(* Logix 5000 project; controller cal1615 1756-L62 rev 20.19; software revision 20.05; part 7 of 81 *)

   p23r11_permissive_jog : BOOL := 1;   // Impreg Servo Operator Side Perimssive Jog
   p23r11_pos_offset : REAL := 0.0005;
   p23r11_request_jog_fwd : BOOL;   // Impreg Servo Operator Side Requset Jog Forward
   p23r11_request_jog_rev : BOOL;   // Impreg Servo Operator Side Requset Jog Reverse
   p23r11_request_position : BOOL;   // Impreg Servo Operator Side Request Position
   p23r11_request_start : BOOL;   // Impreg Servo Operator Side Request Start
   p23r11_request_zero : BOOL;   // Impreg Servo Operator Side Request Zero
   p23r11_selected_position : REAL := 0.016;
   p23r11_servo_not_ready : BOOL;   // Impreg Servo Operator Side Not Ready
   p23r11_servo_status_ab : BOOL := 1;   // Impreg Servo Operator Side AB Status
   p23r11_servo_status_af : BOOL;   // Impreg Servo Operator Side AF Status
   p23r11_servo_status_bb : BOOL;   // Impreg Servo Operator Side BB Status
   p23r11_step_4_dwell : TIMER := (PRE := 1000);
   p23r11_timer : TIMER[4] := ([0].ACC := 33, [0].EN := 1, [0].DN := 1);   // Impreg Servo Operator Side Timer
   p23r11_timer_fault : TIMER[4];   // Impreg Servo Drive Side Fault Delay
   p23r11_timer_warning : TIMER[4];   // Impreg Servo Drive Side Warning Delay
   p23r12 : routine := (comment := -1073741570, state := 3);   // Impreg Servo Drive Side
        .FAULT.0   // Impreg Servo Drive Side Operating Mode Error
        .FAULT.1   // Impreg Servo Drive Side Servo Fault
        .FAULT.3   // Tension Stand 2 VFD Not in Network Mode
        .WARNING.0   // Impreg Servo Drive Side Servo Warning
        .WARNING.1   // Tension Stand 2 VFD Motor Thermistor Not OK
        .WARNING.2   // Tension Stand 2 VFD Motor Blower Not Running
        .WARNING.3   // Tension Stand 2 VFD Brake Thermistor Not Ok
        .UNACK_FAULT   // Impreg Servo Drive Side Unacknoledged Faults Exist
        .UNACK_WARNING   // Impreg Servo Drive Side Unack. Warnings Exist
   p23r12_gap_sequence_enabled : BOOL;
   p23r12_impreg_gap_ds : REAL := 0.016;
   p23r12_offsets : REAL[100] := ([5] := -0.0005, [8] := 0.00015, [10] := -0.0002);
   p23r12_permissive_jog : BOOL := 1;   // Impreg Servo Drive Side Perimssive Jog
   p23r12_pos_offset : REAL;
   p23r12_request_jog_fwd : BOOL;   // Impreg Servo Drive Side Requset Jog Forward
   p23r12_request_jog_rev : BOOL;   // Impreg Servo Drive Side Requset Jog Reverse
   p23r12_request_position : BOOL;   // Impreg Servo Drive Side Request Position
   p23r12_request_start : BOOL;   // Caoter Servo Drive Side Start Request
   p23r12_request_zero : BOOL;   // Impreg Servo Drive Side Request Zero
   p23r12_selected_position : REAL := 0.016;
   p23r12_servo_not_ready : BOOL;   // Impreg Servo Drive Side Not Ready
   p23r12_servo_status_ab : BOOL := 1;   // Impreg Servo Drive Side AB Status
   p23r12_servo_status_af : BOOL;   // Impreg Servo Drive Side AF Status
   p23r12_servo_status_bb : BOOL;   // Impreg Servo Drive Side BB Status
   p23r12_step_4_dwell : TIMER := (PRE := 1000);
   p23r12_timer : TIMER[4] := ([0].ACC := 33, [0].EN := 1, [0].DN := 1);   // Impreg Servo Drive Side Timer
   p23r12_timer_fault : TIMER[4];   // Impreg Servo Drive Side Fault Delay
   p23r12_timer_warning : TIMER[4];   // Impreg Servo Drive Side Warning Delay
   p23r13 : routine := (comment := -1073741697, oneshot := 3);
        .FAULT.0   // Impreg Supply VFD Drive Faulted
        .FAULT.2   // Impreg Supply VFD Drive Not Ready
        .FAULT.3   // Impreg Supply VFD Not in Remote Mode
        .FAULT.4   // Impreg Supply VFD Motor Temperature
        .FAULT_ACK   // Impreg Static Control 2 Faults
        .WARNING.0   // Impreg Supply Fan VFD Drive Warning
        .WARNING.1   // Impreg Supply Fan VFD Supply Filter Dirty
        .WARNING_ACK   // Impreg Static Control 2 Warnings
        .UNACK_FAULT   // Impreg Static Control 2 Unack. Faults Exist
        .UNACK_WARNING   // Impreg Static Control 2 Unack. Warnings Exist
   p23r13_pb_start : BOOL;   // Impreg Supply VFD Start
   p23r13_pb_stop : BOOL;   // Impreg Supply VFD Stop
   p23r13_request_auto_run : BOOL;   // Impreg Supply Fan VFD Request Auto Run
   p23r13_run_permissive : BOOL := 1;   // Impreg Supply VFD Run Permissive
   p23r13_timer_fault : TIMER[10] := ([5].PRE := 5000);   // Impreg Supply VFD Fault Dwell Timer
   p23r13_timer_warning : TIMER[4] := ([1].PRE := 1000, [2].PRE := 10000);   // Impreg Supply VFD Warning Dwell Timer
   p23r13_vfd_stopped : BOOL := 1;   // Impreg Supply VFD Stopped
   p23r15 : routine := (comment := -1073741713, warning := 1, unack_warning := 1);   // Impreg Metering Roll VFD
        .FAULT.0   // Impreg Metering Roll VFD Drive Fault
        .FAULT.2   // Impreg Metering Roll VFD Not Ready
        .FAULT.3   // Impreg Metering Roll VFD Not in Network Mode
        .FAULT.4   // Impreg Metering Roll VFD Motor Temperature Failure
        .WARNING.0   // Impreg Metering VFD Drive Warning
        .WARNING.1   // Impreg Metering Roll VFD Motor Thermistor Not OK
        .WARNING.2   // Impreg Metering Roll VFD Motor Blower Not Running
        .WARNING.3   // Impreg Metering Roll VFD Brake Thermistor Not Ok
        .UNACK_FAULT   // Impreg Metering Roll VFD Unacknoledged Faults Exists
        .UNACK_WARNING   // Impreg Metering Roll VFD Unacknoledged Warning Exists
   p23r15_acc_decel_ramp : SYS_ACC_DEC_RAMP := (IN_param_master_accel_rate := 15.0, IN_param_master_decel_rate := 15.0, IN_last_scan_s := 0.033662);   // Impreg Metering Roll VFD Accel/Decel Ramp
   p23r15_adjust_dwell1 : TIMER := (PRE := 20000);   // Impreg Metering Roll VFD Adjustment Dwell Timer
   p23r15_average_tension : REAL := 87.4577;   // Impreg Metering Roll VFD Average Tension
   p23r15_dead_band_minus : REAL := 45.0;   // Impreg Metering Roll VFD Dead Band -
   p23r15_dead_band_plus : REAL := 55.0;   // Impreg Metering Roll VFD Dead Band +
   p23r15_dead_band_setpoint : REAL := 5.0;
   p23r15_debounce_timer : TIMER := (PRE := 2000, EN := 1, DN := 1);   // Impreg Metering Roll VFD Tension Ok Debounce Timer
   p23r15_ffl : CONTROL := (LEN := 10, POS := 9);   // Impreg Metering Roll VFD Avererage FFL
   p23r15_ffu_temp : REAL := 102.55185;
   p23r15_fll_stack : REAL[50] := ([0] := 98.387886, [1] := 74.37622, [2] := 97.50486, [3] := 91.988014, [4] := 72.294235, [5] := 89.74401, [6] := 102.07388, [7] := 75.97214, [8] := 84.77803, [10] := 108.79131, [11] := 101.68503, [12] := 100.24141, [13] := 100.53305, [14] := 105.432594, [15] := 103.07518, [16] := 106.29294, [17] := 103.507774, [18] := 102.11763, [20] := 103.94038, [21] := 99.57064, [22] := 100.149055, [23] := 101.106606, [24] := 99.040825, [25] := 99.71646, [26] := 98.370056, [27] := 101.34964, [28] := 96.83409, [29] := 100.43584, [30] := 96.83409, [31] := 98.60823, [32] := 99.90603, [33] := 99.76507, [34] := 101.53921, [35] := 98.60823, [36] := 102.02042, [37] := 100.917046, [38] := 106.676926);
   p23r15_mean_adjust_acitve : BOOL;   // Impreg Metering Roll VFD Mean Adjust Active
   p23r15_minus_adjust : REAL := 1.0;
   p23r15_minus_adjust_acitve : BOOL;   // Impreg Metering Roll VFD Minus Adjust Active
   p23r15_minus_offset : REAL := -0.48000002;
   p23r15_neutral_offset : REAL := 0.4;
   p23r15_permissive_jog : BOOL := 1;   // Impreg Impreg VFD Permissive Jog
   p23r15_permissive_run : BOOL := 1;   // Impreg Metering Roll VFD Permissive Run
   p23r15_pid_tension_control : BOOL := 1;   // Impreg Metering Roll VFD PID Wet Web Active
   p23r15_plus_adjust : REAL := 1.0;
   p23r15_plus_adjust_acitve : BOOL;   // Impreg Plus Adjust Active
   p23r15_plus_offset : REAL := 4.7999997;
   p23r15_request_jog_fwd : BOOL;   // Impreg Metering Roll VFD Request Jog FWD
   p23r15_request_jog_rev : BOOL;   // Impreg Metering Roll VFD Request Jog REV
   p23r15_request_line_run : BOOL;   // Impreg Metering Roll VFD Request Line Run
   p23r15_request_thread_fwd : BOOL;   // Impreg Metering Roll VFD Request Thread FWD
   p23r15_request_thread_rev : BOOL;   // Impreg Metering Roll VFD Request Thread REV
   p23r15_sample_timer : TIMER := (PRE := 100);   // Impreg Metering Roll Sample Timer
   p23r15_selected_speed : REAL;   // Impreg Metering Roll VFD Selected Speed
   p23r15_timer_fault : TIMER[10];   // Impreg Pick Up Roll VFD Fault Timer
   p23r15_timer_warning : TIMER[5];   // Impreg Pick Up Roll VFD Warning Timer
   p23r15_ts1_tension_ok : BOOL := 1;   // Impreg Metering Roll VFD TS 1 Tension Ok
   p23r15_zero_speed : BOOL := 1;   // Impreg Metering Roll VFD At Zero Speed
   p23r17_adjusted_speed : REAL;
   p23r17_di_brake : BOOL;
   p23r17_di_therm : BOOL;
   p23r17_permissive_jog : BOOL := 1;
   p23r17_permissive_run : BOOL := 1;
   p23r17_request_jog_fwd : BOOL;
   p23r17_request_thread_fwd : BOOL;
   p23r17_request_thread_rev : BOOL;
   p23r17_selected_speed : REAL;
   p23r17_spd_adj : REAL := -0.5;
   p23r17_sprng_assist_hmi_auto : BOOL;
   p23r17_sprng_assist_hmi_jog : BOOL;
   p23r17_timer_fault : TIMER[10] := ([2].PRE := 3000, [4].ACC := 33, [4].EN := 1, [4].DN := 1, [5].ACC := 33, [5].EN := 1, [5].DN := 1);
   p23r17_timer_warning : TIMER[5];
   p23r17_zero_speed : BOOL := 1;
   p24_di_edge_guide_auto : BOOL := 1;   // Edge Control Inputs SS: Edge Guide Manual/Auto Auto
   p24_di_edge_guide_center : BOOL := 1;   // Edge Control Inputs PB: Edge Guide Center
   p24_di_edge_guide_left : BOOL := 1;   // Edge Control Inputs PB: Edge Guide Left
   p24_di_edge_guide_right : BOOL := 1;   // Edge Control Inputs PB: Edge Guide Right
   p24_dint_to_hmi : DINT[16];
   p24_do_edge_guide_input_1 : BOOL := 1;   // Edge Guide Digital Output Input 1
   p24_do_edge_guide_input_2 : BOOL;   // Edge Guide Digital Output Input 2
   p24_do_edge_guide_input_3 : BOOL;   // Edge Guide Digital Output Input 3
   p24_do_edge_guide_input_4 : BOOL;   // Edge Guide Digital Output Input 4
   p24_do_edge_guide_input_5 : BOOL;   // Edge Guide Digital Output Input 5
   p24_real_to_hmi : REAL[112];   // Tension Stand 2 Real to HMI
   p24r01 : routine := (comment := 7);
   p24r02 : routine := (comment := -1073741761);   // Edge Control Misc Control
        .UNACK_FAULT   // Edge Control Misc Control Unacknowleged Fault Exist
        .UNACK_WARNING   // Edge Control Misc Control Unacknowleged Warning Exist
   p24r02_fault_exists : BOOL;
   p24r02_timer_fault : TIMER[4];   // Edge Control Misc Control Fault Delay
   p24r02_timer_warning : TIMER[4];   // Edge Control Misc Control Warning Delay
   p24r02_unack_fault : BOOL;   // Tension Stand 2 Misc Control Unacknowledged Fault Exists
   p24r02_unack_warning : BOOL;   // Tension Stand 2 Misc Control Unacknowledged Warning Exists
   p24r02_warning_exists : BOOL;
   p24r03 : routine := (comment := -1073741761);   // Edge Control Inputs
        .UNACK_FAULT   // Edge Control Inputs Unacknowleged Fault Exist
        .UNACK_WARNING   // Edge Control Inputs Unacknowleged Warning Exist
   p24r03_timer_fault : TIMER[4];   // Edge Control Inputs Fault Delay
   p24r03_timer_warning : TIMER[4];   // Edge Control Inputs Warning Delay
   p24r04 : routine := (comment := -1073741809);   // Edge Control Outputs
        .UNACK_FAULT   // Edge Control Outputs Unacknowleged Fault Exist
        .UNACK_WARNING   // Edge Control Outputs Unacknowleged Warning Exist
   p24r04_timer_fault : TIMER[4];   // Edge Control Outputs Fault Delay
   p24r04_timer_warning : TIMER[4];   // Edge Control Outputs Warning Dwell
   p24r05 : routine := (comment := -1073741809);   // Edge Control Dint to HMI
        .UNACK_FAULT   // Edge Control Dint to HMI Unacknowleged Fault Exist
        .UNACK_WARNING   // Edge Control Dint to HMI Unacknowleged Warning Exist
   p24r05_timer_fault : TIMER[4];   // Edge Control Dint to HMI Fault Dwell
   p24r05_timer_warning : TIMER[4];   // Edge Control Dint to HMI Warning Delay
   p24r06 : routine := (comment := -1073741793);   // Edge Control Real to HMI
        .UNACK_FAULT   // Edge Control Real to HMI Unacknowleged Fault Exist
        .UNACK_WARNING   // Edge Control Real to HMI Unacknowleged Warning Exist
   p24r06_timer_fault : TIMER[4];   // Edge Control Real to HMI Fault Delay
   p24r06_timer_warning : TIMER[4];   // Edge Control Real to HMI Warning Delay
   p24r07 : routine := (comment := -1073741761);   // Edge Control Alarms
        .UNACK_FAULT   // Edge Control Alarms Unacknowleged Fault Exist
        .UNACK_WARNING   // Edge Control Alarms Unacknowleged Warning Exist
   p24r07_timer_fault : TIMER[4];   // Edge Control Alarms Fault Delay
   p24r07_timer_warning : TIMER[4];   // Edge Control Alarms Warning Delay
   p24r08 : routine := (comment := -1073741761);   // Edge Control Warings
        .UNACK_FAULT   // Edge Control Warnings Unacknowleged Fault Exist
        .UNACK_WARNING   // Edge Control Warnings Unacknowleged Warning Exist
   p24r08_timer_fault : TIMER[4];   // Edge Control Warnings Fault Delay
   p24r08_timer_warning : TIMER[4];   // Edge Control Warnings Warning Delay
   p24r09 : routine := (comment := -1073741761);   // Tension Stand 2 Modes
        .WARNING.1   // Tension Stand 2 Modes Tension Stand in Thread Mode
   p24r09_timer_fault : TIMER[4];   // Edge Control Modes Fault Delay
   p24r09_timer_warning : TIMER[4];   // Edge Control Modes Warning Delay
   p24r10 : routine := (comment := -1073741761);   // Edge Control Edge Guide
        .UNACK_FAULT   // Edge Control Edge Guide Unacknowleged Fault Exist
        .UNACK_WARNING   // Edge Control Edge Guide Unacknowleged Warning Exist
   p24r10_edge_guide_auto_request : BOOL := 1;   // Edge Control Edge Guide Auto Request
   p24r10_edge_guide_center_request : BOOL;   // Edge Control Edge Guide Center Request
   p24r10_edge_guide_jog_left_request : BOOL;   // Edge Control Edge Guide Jog Left Request
   p24r10_edge_guide_jog_right_request : BOOL;   // Edge Control Edge Guide Jog Right Request
   p24r10_timer_fault : TIMER[4];   // Edge Control Edge Guide Fault Delay
   p24r10_timer_warning : TIMER[4];   // Edge Control Edge Guide Warning Delay
   p25_ai_amps : DINT;   // Tension Stand 2 Analog Input TS 2 Motor Current
   p25_ai_hz : DINT;   // Tension Stand 2 Analog Input TS 2 Motor Hertz
   p25_ai_rpm : REAL;
   p25_ai_speed : REAL;   // Tension Stand 2 Inputs Sufrace Speed [fpm]
   p25_ai_torque : REAL;
   p25_ai_ts2_lc : REAL := 122.24563;   // System Metering Roll VFD Minimum Start Tension
   p25_ao_selected_speed : REAL;   // Tension Stand 2 VFD Selected Speed
   p25_ao_torque : REAL := 300.0;
   p25_ao_vfd : REAL;
   p25_control_word : INT := 2#0000_0100_0000_0111;
   p25_di_brake : BOOL := 1;   // Tension Stand 2 Digital Input TS2 & Slitter Brake Temperature OK
   p25_di_jog : BOOL;   // Tension Stand 2 Digital Input SS: Jog
   p25_di_jog_fwd : BOOL;   // Tension Stand 2 Digital Input PB: Jog Forward
   p25_di_jog_rev : BOOL;   // Tension Stand 2 Digital Input PB: Jog Reverse
   p25_di_run : BOOL := 1;   // Tension Stand 2 Digital Input SS: Run
   p25_di_therm : BOOL := 1;   // Tension Stand 2 Digital Input Motor Temperature OK
   p25_di_ts2 : acs800_di_normal := (ready := 1, ctrl_from_net := 1, ref_from_net := 1, at_reference := 1);   // Tension Stand 2 Digital Inputs VFD Inputs
   p25_dint_to_hmi : DINT[16] := ([0] := 983808, [1] := 4915, [4] := 4, [6] := 131072, [7] := 2);   // Tension Stand 2 Dint to HMI
        [0].8   // Tension Stand 2 Dint to HMI Motor Temperature Ok
        [0].9   // Tension Stand 2 Dint to HMI Brake Temperature Ok
        [0].12   // Tension Stand 2 Dint to HMI VFD Faulted
        [0].13   // Tension Stand 2 Dint to HMI VFD Warning
        [0].14   // Tension Stand 2 Dint to HMI VFD Running Forward
        [0].15   // Tension Stand 2 Dint to HMI VFD Running Reverse
        [0].16   // Tension Stand 2 Dint to HMI VFD Ready
        [0].17   // Tension Stand 2 Dint to HMI VFD Control From Net
        [0].18   // Tension Stand 2 Dint to HMI VFD Reference From Net
        [0].19   // Tension Stand 2 Dint to HMI VFD At Reference
        [2].0   // Tension Stand 2 Alarms A00: VFD Drive Faulted
        [2].1   // Tension Stand 2 Alarms A01:
        [2].2   // Tension Stand 2 Alarms A02: VFD Drive Not Ready
        [2].3   // Tension Stand 2 Alarms A03: VFD Drive Not in Remote Mode
        [2].4   // Tension Stand 2 Alarms A04: Motor Temperature
        [2].5   // Tension Stand 2 Alarms A05: Brake Temperature
        [2].6   // Tension Stand 2 Alarms A06:
        [2].7   // Tension Stand 2 Alarms A07:
        [2].8   // Tension Stand 2 Alarms A08:
        [2].9   // Tension Stand 2 Alarms A09:
        [2].10   // Tension Stand 2 Alarms A10:
        [2].11   // Tension Stand 2 Alarms A11:
        [2].12   // Tension Stand 2 Alarms A12:
        [2].13   // Tension Stand 2 Alarms A13:
        [2].14   // Tension Stand 2 Alarms A14:
        [2].15   // Tension Stand 2 Alarms A15:
        [2].16   // Tension Stand 2 Alarms A16:
        [2].17   // Tension Stand 2 Alarms A17:
        [2].18   // Tension Stand 2 Alarms A18:
        [2].19   // Tension Stand 2 Alarms A19:
        [2].20   // Tension Stand 2 Alarms A20:
        [2].21   // Tension Stand 2 Alarms A21:
        [2].22   // Tension Stand 2 Alarms A22:
        [2].23   // Tension Stand 2 Alarms A23:
        [2].24   // Tension Stand 2 Alarms A24:
        [2].25   // Tension Stand 2 Alarms A25:
        [2].26   // Tension Stand 2 Alarms A26:
        [2].27   // Tension Stand 2 Alarms A27:
        [2].28   // Tension Stand 2 Alarms A28:
        [2].29   // Tension Stand 2 Alarms A29:
        [2].30   // Tension Stand 2 Alarms A30:
        [2].31   // Tension Stand 2 Alarms A31:
        [4].0   // Tension Stand 2 Warning W00: VFD Drive Warning
        [4].1   // Tension Stand 2 Warning W01:
        [4].2   // Tension Stand 2 Warning W02:
        [4].3   // Tension Stand 2 Warning W03:
        [4].4   // Tension Stand 2 Warning W04: Tension Stand Not in Run Mode
        [4].5   // Tension Stand 2 Warning W05:
        [4].6   // Tension Stand 2 Warning W06:
        [4].7   // Tension Stand 2 Warning W07:
        [4].8   // Tension Stand 2 Warning W08:
        [4].9   // Tension Stand 2 Warning W09:
        [4].10   // Tension Stand 2 Warning W10:
        [4].11   // Tension Stand 2 Warning W11:
        [4].12   // Tension Stand 2 Warning W12:
        [4].13   // Tension Stand 2 Warning W13:
        [4].14   // Tension Stand 2 Warning W14:
        [4].15   // Tension Stand 2 Warning W15:
        [4].16   // Tension Stand 2 Warning W16:
        [4].17   // Tension Stand 2 Warning W17:
        [4].18   // Tension Stand 2 Warning W18:
        [4].19   // Tension Stand 2 Warning W19:
        [4].20   // Tension Stand 2 Warning W20:
        [4].21   // Tension Stand 2 Warning W21:
        [4].22   // Tension Stand 2 Warning W22:
        [4].23   // Tension Stand 2 Warning W23:
        [4].24   // Tension Stand 2 Warning W24:
        [4].25   // Tension Stand 2 Warning W25:
        [4].26   // Tension Stand 2 Warning W26:
        [4].27   // Tension Stand 2 Warning W27:
        [4].28   // Tension Stand 2 Warning W28:
        [4].29   // Tension Stand 2 Warning W29:
        [4].30   // Tension Stand 2 Warning W30:
        [4].31   // Tension Stand 2 Warning W31:
   p25_param_payout_speed_factor : REAL := 0.2;   // Tension Stand 2 Accumulator Payout Winder Overspeed Factor 0.20 = 1.20 x Line Speed
   p25_param_ts2_jog_speed : REAL := 8.0;   // System Parameter Tension Stand 2 Jog Speed
   p25_real_to_hmi : REAL[112] := ([0] := 122.22771, [40] := 1.0, [41] := 1.0);   // Tension Stand 2 Real to HMI
   p25_status_word : INT := 2#0001_0011_0011_0011;
   p25_ts2_acc_rate : REAL := 8.0;
   p25_ts2_decel_rate : REAL := 8.0;
   p25_ts2_gear_ratio : REAL := 108.75;
   p25_ts2_roll_diameter_ft : REAL := 1.0;
   p25_ts2_vfd : ABB_PROTOCOL_VFD := (STATUS_WORD := 4915, CONTROL_WORD := 1031, IN_DRIVE_PERMISSIVE := 1);
   p25_vfd_input_max : REAL := 2000.0;
   p25_vfd_input_min : REAL := -2000.0;
   p25_vfd_output_max : REAL := 20000.0;
   p25_vfd_output_min : REAL := -20000.0;
   p25r01 : routine := (comment := 7);
   p25r02 : routine := (comment := -1073741761);
        .UNACK_FAULT   // Tension Stand 2 Misc Control Unacknowleged Faults Exist
        .UNACK_WARNING   // Tension Stand 2 Misc Control Unacknowleged Warnings Exist
   p25r02_fault_exists : BOOL;
   p25r02_tension_dev_max : REAL := 66.0;
   p25r02_tension_dev_min : REAL := 54.0;
   p25r02_timer_fault : TIMER[4];   // Tension Stand 2 Misc Control Fault Dwell Timer
   p25r02_timer_warning : TIMER[4];   // Tension Stand 2 Misc Control Warning Dwell Timer
   p25r02_unack_fault : BOOL;   // Upper Poly Letoff Misc Control Unacknowledged Fault Exists
   p25r02_unack_warning : BOOL;   // Upper Poly Letoff Misc Control Unacknowledged Warning Exists
   p25r02_warning_exists : BOOL := 1;
   p25r03 : routine := (comment := -1073741761);
        .UNACK_FAULT   // Tension Stand 2 Input Unacknowleged Faults Exist
        .UNACK_WARNING   // Tension Stand 2 Input Unacknowleged Warnings Exist
   p25r03_ave_tq : REAL;
   p25r03_hz : SYS_SCP := (Input_Max := 2000.0, Output_Max := 60.0);   // Tension Stand 2 Analog Inputs SCP Hz
   p25r03_lc_input_max : REAL := 30860.0;
   p25r03_lc_input_min : REAL;
   p25r03_lc_output_max : REAL := 250.0;
   p25r03_lc_output_min : REAL;
   p25r03_lc_scp : SYS_SCP := (Input := 15110.0, Input_Max := 30860.0, Output_Max := 250.0, Output := 122.40765);   // Tension Stand 2 Analog Input Load Cell Scaling
   p25r03_sample_timer : TIMER := (PRE := 200, ACC := 164, EN := 1, TT := 1);
   p25r03_scaled_vfd_in : REAL;
   p25r03_timer_fault : TIMER[4];   // Tension Stand 2 Inputs Fault Dwell Timer
   p25r03_timer_warning : TIMER[4];   // Tension Stand 2 Inputs Warning Dwell Timer
   p25r03_tq_ave_ctrl : CONTROL := (LEN := 19);
   p25r03_tq_buffer : REAL[20];
   p25r03_tq_fifo : CONTROL := (LEN := 20, POS := 20, DN := 1);
   p25R03_ts2_vfd_rpm_to_speed : SYS_RPM_TO_SPEED := (IN_gear_ratio := 108.75, IN_roll_diameter := 1.0);   // Tension Stand 2 Analog Input VFD RPM to Roll Surface Speed
   p25r03_unload : DINT;
   p25r03_vfd_in_scaling : SYS_SCP := (Input_Min := -20000.0, Input_Max := 20000.0, Output_Min := -2000.0, Output_Max := 2000.0);
   p25r03_vfd_input_max : REAL := 20000.0;
   p25r03_vfd_input_min : REAL := -20000.0;
   p25r03_vfd_out_scaling : SYS_SCP := (Input_Min := -2000.0, Input_Max := 2000.0, Output_Min := -20000.0, Output_Max := 20000.0);
   p25r03_vfd_output_max : REAL := 2000.0;
   p25r03_vfd_output_min : REAL := -2000.0;
   p25r04 : routine := (comment := -1073741761);
        .UNACK_FAULT   // Tension Stand 2 Output Unacknowleged Faults Exist
        .UNACK_WARNING   // Tension Stand 2 Output Unacknowleged Warnings Exist
   p25r04_speed_to_vfd_ts2_scp : SYS_SPEED_TO_VFD := (IN_gear_ratio := 108.75, IN_roll_diameter := 1.0);   // Tension Stand 2 Outputs Speed to Tension Stand 2 VFD
   p25r04_timer_fault : TIMER[4];   // Tension Stand 2 Outputs Fault Dwell Timer
   p25r04_timer_warning : TIMER[4];   // Tension Stand 2 Outputs Warning Dwell Timer
   p25r05 : routine := (comment := -1073741761);
        .UNACK_FAULT   // Tension Stand 2 Dint to HMI Unacknowleged Faults Exist
        .UNACK_WARNING   // Tension Stand 2 Dint to HMI Unacknowleged Warnings Exist
   p25r05_timer_fault : TIMER[4];   // Tension Stand 2 Dint to HMI Fault Dwell Timer
   p25r05_timer_warning : TIMER[4];   // Tension Stand 2 Dint to HMI Warning Dwell Time
   p25r06 : routine := (comment := -1073741572);
        .UNACK_FAULT   // Tension Stand 2 Real to HMI Unacknowleged Faults Exist
        .UNACK_WARNING   // Tension Stand 2 Real to HMI Unacknowleged Warnings Exist
   p25r06_ave_lc : REAL := 122.29934;
   p25r06_lc_ave_ctrl : CONTROL := (LEN := 19);
   p25r06_lc_buffer : REAL[20] := ([0] := 122.16462, [1] := 122.002594, [2] := 122.32664, [3] := 122.40765, [4] := 122.24563, [5] := 122.0836, [6] := 122.16462, [7] := 122.0836, [8] := 122.002594, [9] := 122.48056, [10] := 122.40765, [11] := 122.16462, [12] := 122.24563, [13] := 122.0836, [14] := 122.0836, [15] := 122.0836, [16] := 122.16462, [17] := 122.32664, [18] := 122.32664, [19] := 122.32664);
   p25r06_lc_ctrl : CONTROL := (LEN := 20, POS := 20, DN := 1);
   p25r06_sample_timer : TIMER := (PRE := 200, ACC := 65, EN := 1, TT := 1);
   p25r06_timer_fault : TIMER[4];   // Tension Stand 2 Real to HMI Fault Dwell Timer
   p25r06_timer_warning : TIMER[4];   // Tension Stand 2 Real to HMI Warning Dwell Timer
   p25r06_unload : REAL := 122.24563;
   p25r07 : routine := (comment := -1073741761);
        .UNACK_FAULT   // Tension Stand 2 Alarms Unacknowleged Faults Exist
        .UNACK_WARNING   // Tension Stand 2 Alarms Unacknowleged Warnings Exist
   p25r07_timer_fault : TIMER[4];   // Tension Stand 2 Alarms Fault Dwell Time
   p25r07_timer_warning : TIMER[4];   // Tension Stand 2 Alarms Warning Dwell Timer
   p25r08 : routine := (comment := -1073741761);
        .WARNING.0   // Tension Stand 2 Modes Tension Stand Not in Run Mode
        .WARNING.1   // Tension Stand 2 Modes Tension Stand in Thread Mode
        .UNACK_FAULT   // Tension Stand 2 Warnings Unacknowleged Faults Exist
        .UNACK_WARNING   // Tension Stand 2 Warnings Unacknowleged Warnings Exist
   p25r08_timer_fault : TIMER[4];   // Tension Stand 2 Warnings Fault Dwell Timer
   p25r08_timer_warning : TIMER[4];   // Tension Stand 2 Warnings Warning Dwell Timer
   p25r09 : routine := (comment := -1073741761);   // Upper Poly Letoff Modes
        .UNACK_FAULT   // Tension Stand 2 Modes Unacknowleged Faults Exist
        .UNACK_WARNING   // Tension Stand 2 Modes Unacknowleged Warnings Exist
   p25r09_mode_jog : BOOL;   // Tension Stand 2 Modes Jog Mode
   p25r09_mode_run : BOOL := 1;   // Tension Stand 2 Modes Run Mode
   p25r09_mode_thread : BOOL;   // Tension Stand 2 Modes Thread Mode
   p25r09_pb_jog_fwd : BOOL;   // Tension Stand 2 Modes PB: Jog Forward
   p25r09_pb_jog_rev : BOOL;   // Tension Stand 2 Modes PB: Jog Reverse
   p25r09_timer_fault : TIMER[4];   // Tension Stand 2 Modes Fault Dwell Timer
   p25r09_timer_warning : TIMER[4];   // Tension Stand 2 Modes Warning Dwell Timer
   p25r10 : routine := (comment := -1073741761);
        .UNACK_FAULT   // Tension Stand 2 Speed Unacknowleged Faults Exist
        .UNACK_WARNING   // Tension Stand 2 Speed Unacknowleged Warnings Exist
   p25r10_calc_speed_offset : REAL;
   p25r10_param_psn_gain : REAL := 15.0;   // Tension Stand 2 Parameter Position Gain
   p25r10_pid_manual_request : BOOL := 1;
   p25r10_pid_out : REAL := 50.0;
   p25r10_pid_psn : PID := (CTL := -2078243712, EN := 1, SWM := 1, NOBC := 1, INI := 1, DVNA := 1, PVHA := 1, SP := 60.0, KP := 1.0, KI := 1.0, BIAS := 1.0, MAXS := 500.0, SO := 50.0, MAXO := 100.0, UPD := 0.01, PV := 122.32664, ERR := -62.326637, OUT := 50.0, MAXI := 500.0, MAXCV := 100.0, MAXTIE := 100.0, DATA[0] := 61.46533, DATA[1] := -391.44525, DATA[2] := 122.32664, DATA[3] := -62.326637, DATA[4] := 60.0, DATA[5] := 0.2, DATA[6] := 1.0, DATA[7] := 0.16, DATA[8] := 1.0, DATA[9] := 1.0, DATA[11] := 1.0, DATA[12] := 1.0, DATA[15] := 1.0, DATA[16] := 1.0);   // Tension Stand 2 Speed Tension PID Dancer Position Process Variable
   p25r10_pid_psn_cv : REAL := 50.0;
   p25r10_pid_psn_pv : REAL := 122.0836;   // Tension Stand 2 Speed Tension PID Dancer Position Process Variable
   p25r10_speed_offset : REAL;   // Tension Stand 2 Speed tension Speed Offset from Base
   p25r10_tension_request : BOOL;
   p25r10_timer_fault : TIMER[4];   // Tension Stand 2 Speed Tension Fault Dwell Timer
   p25r10_timer_warning : TIMER[4];   // Tension Stand 2 Speed Tension Warning Dwell Timer
   p25r11 : routine := (comment := -1073741713, warning := 4, warning_ack := 4);   // Tension Stand 2 VFD
        .FAULT.0   // Tension Stand 2 VFD Drive Faulted
        .FAULT.2   // Tension Stand 2 VFD Drive Not Ready
        .FAULT.3   // Tension Stand 2 VFD Drive Not in Remote Mode
        .FAULT.4   // Tension Stand 2 VFD Motor Temperature
        .FAULT.5   // Tension Stand 2 VFD Brake Temperature
        .WARNING   // Tension Stand 2 VFD
        .WARNING.0   // Tension Stand 2 VFD Drive Warning
        .UNACK_FAULT   // Tension Stand 2 VFd Unacknowleged Faults Exist
        .UNACK_WARNING   // Tension Stand 2 VFD Unacknowleged Warnings Exist
   p25r11_acc_decel_ramp : SYS_ACC_DEC_RAMP := (IN_param_master_accel_rate := 8.0, IN_param_master_decel_rate := 8.0, IN_last_scan_s := 0.034268);   // Tension Stand 2 VFD Accel /Decel Ramp
   p25r11_at_zero : BOOL := 1;   // Tension Stand 2 VFD At Zero Speed
   p25r11_permissive_jog_thread : BOOL := 1;   // Tension Stand 2 VFD Permissive Jog/Thread
   p25r11_request_jog_fwd : BOOL;   // Tension Stand 2 VFD Request Jog FWD
   p25r11_request_jog_rev : BOOL;   // Tension Stand 2 VFD Request Jog REV
   p25r11_request_line_jog : BOOL;   // Tension Stand 2 VFD Request Line Jog
   p25r11_request_line_run : BOOL;   // Tension Stant 2 VFD Request Line Run
   p25r11_request_thread_fwd : BOOL;   // Tension Stand 2 VFD Request Thread FWD
   p25r11_request_thread_rev : BOOL;   // Tension Stand 2 VFD Request Thread REV
   p25r11_selected_speed : REAL;   // Tension Stand 2 VFD Selected Speed
   p25r11_timer_fault : TIMER[10];   // Tension Stand 2 VFD Fault Dwell Timer
   p25r11_timer_warning : TIMER[4] := ([1].PRE := 10000, [2].PRE := 10000);   // Tension Stand VFD Warning Dwell Timer
   p25r11_vfd_start_request : BOOL;
   p25r20_pide_cv : REAL := 50.0;
   p26_ao_dia_a : REAL := 22.867153;   // Upper Poly Letoff Analog Input Letoff A Diameter
   p26_ao_dia_b : REAL := 18.7;   // Upper Poly Letoff Analog Input Letoff B Diameter
   p26_dint_to_hmi : DINT[16] := ([0] := 5);   // Upper Poly Letoff Dint to HMI
        [0].0   // Upper Poly Letoff Dint to HMI PI: A Enabled
        [0].2   // Upper Poly Letoff Dint to HMI PI: B Enabled
        [2].0   // Upper Poly Letoff Alarms A00:
        [2].1   // Upper Poly Letoff Alarms A01:
        [2].2   // Upper Poly Letoff Alarms A02:
        [2].3   // Upper Poly Letoff Alarms A03:
        [2].4   // Upper Poly Letoff Alarms A04:
        [2].5   // Upper Poly Letoff Alarms A05:
        [2].6   // Upper Poly Letoff Alarms A06:
        [2].7   // Upper Poly Letoff Alarms A07:
        [2].8   // Upper Poly Letoff Alarms A08:
        [2].9   // Upper Poly Letoff Alarms A09:
        [2].10   // Upper Poly Letoff Alarms A10:
        [2].11   // Upper Poly Letoff Alarms A11:
        [2].12   // Upper Poly Letoff Alarms A12:
        [2].13   // Upper Poly Letoff Alarms A13:
        [2].14   // Upper Poly Letoff Alarms A14:
        [2].15   // Upper Poly Letoff Alarms A15:
        [2].16   // Upper Poly Letoff Alarms A16:
        [2].17   // Upper Poly Letoff Alarms A17:
        [2].18   // Upper Poly Letoff Alarms A18:
        [2].19   // Upper Poly Letoff Alarms A19:
        [2].20   // Upper Poly Letoff Alarms A20:
        [2].21   // Upper Poly Letoff Alarms A21:
        [2].22   // Upper Poly Letoff Alarms A22:
        [2].23   // Upper Poly Letoff Alarms A23:
        [2].24   // Upper Poly Letoff Alarms A24:
        [2].25   // Upper Poly Letoff Alarms A25:
        [2].26   // Upper Poly Letoff Alarms A26:
        [2].27   // Upper Poly Letoff Alarms A27:
        [2].28   // Upper Poly Letoff Alarms A28:
        [2].29   // Upper Poly Letoff Alarms A29:
        [2].30   // Upper Poly Letoff Alarms A30:
        [2].31   // Upper Poly Letoff Alarms A31:
        [4].0   // Upper Poly Letoff Warnings W00
        [4].1   // Upper Poly Letoff Warnings W01:
        [4].2   // Upper Poly Letoff Warnings W02:
        [4].3   // Upper Poly Letoff Warnings W03:
        [4].4   // Upper Poly Letoff Warnings W04:
        [4].5   // Upper Poly Letoff Warnings W05:
        [4].6   // Upper Poly Letoff Warnings W06:
        [4].7   // Upper Poly Letoff Warnings W07:
        [4].8   // Upper Poly Letoff Warnings W08:
        [4].9   // Upper Poly Letoff Warnings W09:
        [4].10   // Upper Poly Letoff Warnings W10:
        [4].11   // Upper Poly Letoff Warnings W11:
        [4].12   // Upper Poly Letoff Warnings W12:
        [4].13   // Upper Poly Letoff Warnings W13:
        [4].14   // Upper Poly Letoff Warnings W14:
        [4].15   // Upper Poly Letoff Warnings W15:
        [4].16   // Upper Poly Letoff Warnings W16:
        [4].17   // Upper Poly Letoff Warnings W17:
        [4].18   // Upper Poly Letoff Warnings W18:
        [4].19   // Upper Poly Letoff Warnings W19:
        [4].20   // Upper Poly Letoff Warnings W20:
        [4].21   // Upper Poly Letoff Warnings W21:
        [4].22   // Upper Poly Letoff Warnings W22:
        [4].23   // Upper Poly Letoff Warnings W23:
        [4].24   // Upper Poly Letoff Warnings W24:
        [4].25   // Upper Poly Letoff Warnings W25:
        [4].26   // Upper Poly Letoff Warnings W26:
        [4].27   // Upper Poly Letoff Warnings W27:
        [4].28   // Upper Poly Letoff Warnings W28:
        [4].29   // Upper Poly Letoff Warnings W29:
        [4].30   // Upper Poly Letoff Warnings W30:
        [4].31   // Upper Poly Letoff Warnings W31:
   p26_inactive_tension_sp : REAL;
   p26_ltf_a_sensor_input_max : REAL := 30959.0;
   p26_ltf_a_sensor_input_min : REAL := 100.0;
   p26_ltf_a_sensor_output_max : REAL := 55.0;
   p26_ltf_a_sensor_output_min : REAL := 4.0;
   p26_ltf_b_sensor_input_max : REAL := 30959.0;
   p26_ltf_b_sensor_input_min : REAL := 100.0;
   p26_ltf_b_sensor_output_max : REAL := 55.0;
   p26_ltf_b_sensor_output_min : REAL := 4.0;
   p26_real_to_hmi : REAL[112] := ([0] := 22.867153, [1] := 18.7);   // Lower Poly Letoff Real to HMI
   p26_ula_prs_input_max : REAL := 20.0;
   p26_ula_prs_input_min : REAL := 3.5;
   p26_ula_prs_output_max : REAL := 30840.0;
   p26_ula_prs_output_min : REAL := 5397.0;
   p26_ulb_prs_input_max : REAL := 20.0;
   p26_ulb_prs_input_min : REAL := 3.5;
   p26_ulb_prs_output_max : REAL := 30840.0;
   p26_ulb_prs_output_min : REAL := 5397.0;
   p26r01 : routine := (comment := 7);   // Upper Poly Letoff
   p26r02 : routine := (comment := -1073741761);   // Upper Poly Letoff
        .UNACK_FAULT   // Upper Poly Letoff Misc Control Unacknoledged Faults Exist
        .UNACK_WARNING   // Upper Poly Letoff Misc Control Unacknoledged Warnings Exist
   p26r02_fault_exists : BOOL;
   p26r02_timer_fault : TIMER[4];   // Upper Poly Letoff Misc Control Fault Delay
   p26r02_timer_warning : TIMER[4];   // Upper Poly Letoff Misc Control Warning Delay
   p26r02_unack_fault : BOOL;   // Upper Poly Letoff Misc Control Unacknowledged Fault Exists
   p26r02_unack_warning : BOOL;   // Upper Poly Letoff Misc Control Unacknowledged Warning Exists
   p26r02_warning_exists : BOOL;
   p26r03 : routine := (comment := -1073741761);   // Upper Poly Letoff Input
        .UNACK_FAULT   // Upper Poly Letoff Input Unacknoledged Faults Exist
        .UNACK_WARNING   // Upper Poly Letoff Inputs Unacknoledged Warnings Exist
   p26r03_a_radius : REAL := 11.41705;
   p26r03_ai_dia_a_sensor : REAL := 4.816423;
   p26r03_ai_dia_b_sensor : REAL := 4.0;
   p26r03_b_radius : REAL := 9.35;
   p26r03_ltf_a_sensor_scp : SYS_SCP := (Input := 604.0, Input_Min := 100.0, Input_Max := 30959.0, Output_Min := 4.0, Output_Max := 55.0, Output := 4.8329496);   // Upper Poly Letoff Analog Input Diameter A Sensor Scaling
   p26r03_ltf_b_sensor_scp : SYS_SCP := (Input := 60.0, Input_Min := 100.0, Input_Max := 30959.0, Output_Min := 4.0, Output_Max := 55.0, Output := 4.0);   // Upper Poly Letoff Analog Input Letoff B Diameter Sensor Scaling
   p26r03_timer_fault : TIMER[4];   // Lower Poly Letoff Input Fault Delay
   p26r03_timer_warning : TIMER[4];   // Lower Poly Letoff Input Warning Delay
   p26r03_upper_A_tension_on : BOOL := 1;
   p26r03_upper_B_tension_on : BOOL := 1;
   p26r03_upper_poly_a_distance : REAL := 16.25;
   p26r03_upper_poly_b_distance : REAL := 13.35;
   p26r04 : routine := (comment := -1073741761);   // Upper Poly Letoff Output
        .UNACK_FAULT   // Upper Poly Letoff Output Unacknoledged Faults Exist
        .UNACK_WARNING   // Upper Poly Letoff Outputs Unacknoledged Warnings Exist
   p26r04_timer_fault : TIMER[4];   // Lower Poly Letoff Output Fault Delay
   p26r04_timer_warning : TIMER[4];   // Lower Poly Letoff Output Warning Delay
   p26r04_ula_prs_scp : SYS_SCP := (Input := 22.867153, Input_Min := 3.5, Input_Max := 20.0, Output_Min := 5397.0, Output_Max := 30840.0, Output := 30840.0);   // Upper Poly Lefoff Analog Output Letoff A Brake Pressure
   p26r04_ulb_prs_scp : SYS_SCP := (Input := 18.7, Input_Min := 3.5, Input_Max := 20.0, Output_Min := 5397.0, Output_Max := 30840.0, Output := 28835.4);   // Upper Poly Lefoff Analog Output Letoff B Brake Pressure
   p26r05 : routine := (comment := -1073741761);   // Upper Poly Letoff Dint to HMI
        .UNACK_FAULT   // Upper Poly Letoff Dint to HMI Unacknoledged Faults Exist
        .UNACK_WARNING   // Upper Poly Letoff Dint to HMI Unacknoledged Warnings Exist
   p26r05_timer_fault : TIMER[4];   // Lower Poly Letoff Dint to HMI Fault Delay
   p26r05_timer_warning : TIMER[4];   // Lower Poly Letoff Dint to HMI Warning Delay
   p26r06 : routine := (comment := -1073741572);   // Upper Poly Letoff Real to HMI
        .UNACK_FAULT   // Upper Poly Letoff Real to HMI Unacknoledged Faults Exist
        .UNACK_WARNING   // Upper Poly Letoff Real to HMI Unacknoledged Warnings Exist
   p26r06_timer_fault : TIMER[4];   // Lower Poly Letoff Real to HMI Fault Delay
   p26r06_timer_warning : TIMER[4];   // Lower Poly Letoff Real to HMI Warning Delay
   p26r07 : routine := (comment := -1073741761);   // Upper Poly Letoff Alarms
        .UNACK_FAULT   // Upper Poly Letoff Alarms Unacknoledged Faults Exist
        .UNACK_WARNING   // Upper Poly Letoff Alarms Unacknoledged Warnings Exist
   p26r07_timer_fault : TIMER[4];   // Lower Poly Letoff Alarms Fault Delay
   p26r07_timer_warning : TIMER[4];   // Lower Poly Letoff Alarms Warning Delay
   p26r08 : routine := (comment := -1073741761);   // Upper Poly Letoff Warnings
        .UNACK_FAULT   // Upper Poly Letoff Warnings Unacknoledged Faults Exist
        .UNACK_WARNING   // Upper Poly Letoff Warnings Unacknoledged Warnings Exist
   p26r08_timer_fault : TIMER[4];   // Upper Poly Letoff Warnings Fault Delay
   p26r08_timer_warning : TIMER[4];   // Upper Poly Letoff Warnings Warning Delay
   p26r09 : routine := (comment := -1073741761);   // Upper Poly Letoff Modes
        .UNACK_FAULT   // Upper Poly Letoff Modes Unacknoledged Faults Exist
        .UNACK_WARNING   // Upper Poly Letoff Modes Unacknoledged Warnings Exist
   p26r09_timer_fault : TIMER[4];   // Lower Poly Letoff Modes Fault Delay
   p26r09_timer_warning : TIMER[4];   // Lower Poly Letoff Modes Warning Delay
   p26r10 : routine := (comment := -1073741777);   // Upper Poly Letoff Tension
        .UNACK_FAULT   // Upper Poly Letoff Tension Unacknoledged Faults Exist
        .UNACK_WARNING   // Upper Poly Letoff Tension Unacknoledged Warnings Exist
   p26r10_timer_fault : TIMER[4];   // Lower Poly Letoff Fault Delay
   p26r10_timer_warning : TIMER[4];   // Lower Poly Letoff Warning Delay
   p26r10_ula_selected_tension : REAL := 2.0;   // Upper Poly Letoff Tension A Selected Tension
   p26r10_ulb_selected_tension : REAL := 2.0;   // Upper Poly Letoff Tension B Selected Tension
   p26r10_unwind_a_brake_torque : REAL := 1.9055961;   // Upper Poly Letoff Tension Letoff A Brake Torque
   p26r10_unwind_a_dia_ft : REAL := 1.9055961;   // Upper Poly Letoff Tension Diameter A [ft]
   p26r10_unwind_b_brake_torque : REAL := 1.5583334;   // Upper Poly Letoff Tension Letoff B Brake Torque
   p26r10_unwind_b_dia_ft : REAL := 1.5583334;   // Upper Poly Letoff Tension Diameter B [ft]
   p27_ao_dia_a : REAL := -13.184677;   // Lower Poly Letoff Analog Input Letoff A Diameter
   p27_ao_dia_b : REAL := -85.238045;   // Lower Poly Letoff Analog Input Letoff B Diameter
   p27_dint_to_hmi : DINT[16] := ([0] := 5);   // Lower Poly Letoff Alarms
        [0].0   // Lower Poly Letoff Dint to HMI PI: A Enabled
        [0].2   // Lower Poly Letoff Dint to HMI PI: B Enabled
        [1].0   // Lower Poly Letoff Dint to HMI Lower Poly Letoff A VFD Faulted
        [1].1   // Lower Poly Letoff Dint to HMI Lower Poly Letoff A VFD Warning
        [1].2   // Lower Poly Letoff Dint to HMI Lower Poly Letoff A VFD Running Forward
        [1].3   // Lower Poly Letoff Dint to HMI Lower Poly Letoff A VFD Running Reverse
        [1].4   // Lower Poly Letoff Dint to HMI Lower Poly Letoff A VFD Ready
        [1].5   // Lower Poly Letoff Dint to HMI Lower Poly Letoff A VFD Control from Net
        [1].6   // Lower Poly Letoff Dint to HMI Lower Poly Letoff A VFD Reference from Net
        [1].7   // Lower Poly Letoff Dint to HMI Lower Poly Letoff A VFD At Reference
        [2].0   // Lower Poly Letoff Alarms A00:
        [2].1   // Lower Poly Letoff Alarms A01:
        [2].2   // Lower Poly Letoff Alarms A02:
        [2].3   // Lower Poly Letoff Alarms A03:
        [2].4   // Lower Poly Letoff Alarms A04:
        [2].5   // Lower Poly Letoff Alarms A05:
        [2].6   // Lower Poly Letoff Alarms A06:
        [2].7   // Lower Poly Letoff Alarms A07:
        [2].8   // Lower Poly Letoff Alarms A08:
        [2].9   // Lower Poly Letoff Alarms A09:
        [2].10   // Lower Poly Letoff Alarms A10:
        [2].11   // Lower Poly Letoff Alarms A11:
        [2].12   // Lower Poly Letoff Alarms A12:
        [2].13   // Lower Poly Letoff Alarms A13:
        [2].14   // Lower Poly Letoff Alarms A14:
        [2].15   // Lower Poly Letoff Alarms A15:
        [2].16   // Lower Poly Letoff Alarms A16:
        [2].17   // Lower Poly Letoff Alarms A17:
        [2].18   // Lower Poly Letoff Alarms A18:
        [2].19   // Lower Poly Letoff Alarms A19:
        [2].20   // Lower Poly Letoff Alarms A20:
        [2].21   // Lower Poly Letoff Alarms A21:
        [2].22   // Lower Poly Letoff Alarms A22:
        [2].23   // Lower Poly Letoff Alarms A23:
        [2].24   // Lower Poly Letoff Alarms A24:
        [2].25   // Lower Poly Letoff Alarms A25:
        [2].26   // Lower Poly Letoff Alarms A26:
        [2].27   // Lower Poly Letoff Alarms A27:
        [2].28   // Lower Poly Letoff Alarms A28:
        [2].29   // Lower Poly Letoff Alarms A29:
        [2].30   // Lower Poly Letoff Alarms A30:
        [2].31   // Lower Poly Letoff Alarms A31:
        [4].0   // Lower Poly Letoff Warnings W00
        [4].1   // Lower Poly Letoff Warnings W01:
        [4].2   // Lower Poly Letoff Warnings W02:
        [4].3   // Lower Poly Letoff Warnings W03:
        [4].4   // Lower Poly Letoff Warnings W04:
        [4].5   // Lower Poly Letoff Warnings W05:
        [4].6   // Lower Poly Letoff Warnings W06:
        [4].7   // Lower Poly Letoff Warnings W07:
        [4].8   // Lower Poly Letoff Warnings W08:
        [4].9   // Lower Poly Letoff Warnings W09:
        [4].10   // Lower Poly Letoff Warnings W10:
        [4].11   // Lower Poly Letoff Warnings W11:
        [4].12   // Lower Poly Letoff Warnings W12:
        [4].13   // Lower Poly Letoff Warnings W13:
        [4].14   // Lower Poly Letoff Warnings W14:
        [4].15   // Lower Poly Letoff Warnings W15:
        [4].16   // Lower Poly Letoff Warnings W16:
        [4].17   // Lower Poly Letoff Warnings W17:
        [4].18   // Lower Poly Letoff Warnings W18:
        [4].19   // Lower Poly Letoff Warnings W19:
        [4].20   // Lower Poly Letoff Warnings W20:
        [4].21   // Lower Poly Letoff Warnings W21:
        [4].22   // Lower Poly Letoff Warnings W22:
        [4].23   // Lower Poly Letoff Warnings W23:
        [4].24   // Lower Poly Letoff Warnings W24:
        [4].25   // Lower Poly Letoff Warnings W25:
        [4].26   // Lower Poly Letoff Warnings W26:
        [4].27   // Lower Poly Letoff Warnings W27:
        [4].28   // Lower Poly Letoff Warnings W28:
        [4].29   // Lower Poly Letoff Warnings W29:
        [4].30   // Lower Poly Letoff Warnings W30:
        [4].31   // Lower Poly Letoff Warnings W31:
        [5].1   // Winder Dint to HMI Liner Winder VFD Warning
        [5].4   // Winder Dint to HMI Liner Winder VFD Ready
        [5].5   // Winder Dint to HMI Liner Winder VFD Control from Net
        [5].6   // Winder Dint to HMI Liner Winder VFD Reference from Net
        [5].7   // Winder Dint to HMI Liner Winder VFD At Reference
   p27_inactive_tension_sp : REAL;   // Lower Poly Letoff Tension Inactive Tension Setpoint
   p27_lft_a_prs_input_max : REAL := 30959.0;
   p27_lft_a_prs_input_min : REAL := 100.0;
   p27_lft_a_prs_output_max : REAL := 55.0;
   p27_lft_a_prs_output_min : REAL := 4.0;
   p27_lft_b_prs_input_max : REAL := 30959.0;
   p27_lft_b_prs_input_min : REAL := 100.0;
   p27_lft_b_prs_output_max : REAL := 55.0;
   p27_lft_b_prs_output_min : REAL := 4.0;
   p27_lla_prs_input_max : REAL := 20.0;
   p27_lla_prs_input_min : REAL := 3.5;
   p27_lla_prs_output_max : REAL := 30840.0;
   p27_lla_prs_output_min : REAL := 5397.0;
   p27_lla_prs_scp : SYS_SCP := (Input := -3.123169, Input_Min := 3.5, Input_Max := 20.0, Output_Min := 5397.0, Output_Max := 30840.0, Output := 5397.0);   // Lower Poly Letoff Analog Output Letoff A Brake Pressure
   p27_llb_prs_input_max : REAL := 20.0;
   p27_llb_prs_input_min : REAL := 3.5;
   p27_llb_prs_output_max : REAL := 30840.0;
   p27_llb_prs_output_min : REAL := 5397.0;
   p27_llb_prs_scp : SYS_SCP := (Input := 16.6, Input_Min := 3.5, Input_Max := 20.0, Output_Min := 5397.0, Output_Max := 30840.0, Output := 25597.201);   // Lower Poly Letoff Analog Output Letoff B Brake Pressure
   p27_real_to_hmi : REAL[112] := ([0] := 54.0, [1] := 16.6);   // Winder Real to HMI
   p27r01 : routine := (comment := 7);   // Winder Main
   p27r02 : routine := (comment := -1073741761);   // Winder Misc Control
        .UNACK_FAULT   // Lower Poly Letoff Misc Control Unacknoledged Fault Exist
        .UNACK_WARNING   // Lower Poly Letoff Misc Control Unacknoledged Warnnings Exist
   p27r02_fault_exists : BOOL;
   p27r02_timer_fault : TIMER[4];   // Winder Misc Control Fault Delay
   p27r02_timer_warning : TIMER[4];   // Winder Misc Control Warning Delay
   p27r02_unack_fault : BOOL;   // Lower Poly Letoff Misc Control Unacknowledged Fault Exists
   p27r02_unack_warning : BOOL;   // Lower Poly Letoff Misc Control Unacknowledged Warning Exists
   p27r02_warning_exists : BOOL;
   p27r03 : routine := (comment := -1073741761);   // Winder Input
        .UNACK_FAULT   // Lower Poly Letoff Input Unacknoledged Fault Exist
        .UNACK_WARNING   // Lower Poly Letoff Inputs Unacknoledged Warnnings Exist
   p27r03_a_radius : REAL := -3.26054;
   p27r03_ai_dia_a_sensor : REAL := 35.09349;   // Letoff Accumulator Final Accumulator Decel
   p27r03_ai_dia_b_sensor : REAL := 54.91902;
   p27r03_b_radius : REAL := -42.619022;   // Lower Poly Letoff Analog Input B Radius
   p27r03_lower_A_tension_on : BOOL := 1;
   p27r03_lower_B_tension_on : BOOL := 1;
   p27r03_ltf_a_diameter_scp : SYS_SCP := (Input := 30870.0, Input_Min := 100.0, Input_Max := 30959.0, Output_Min := 4.0, Output_Max := 55.0, Output := 54.852913);   // Lower Poly Letoff Analog Input Letoff A Diameter
   p27r03_ltf_b_diameter_scp : SYS_SCP := (Input := 60.0, Input_Min := 100.0, Input_Max := 30959.0, Output_Min := 4.0, Output_Max := 55.0, Output := 4.0);   // Lower Poly Letoff Analog Input Letoff B Diameter
   p27r03_timer_fault : TIMER[4];   // Winder Input Fault Delay
   p27r03_timer_warning : TIMER[4];   // Winder Input Warning Delay
   p27r03_winder_a_distance : REAL := 31.0;   // Letoff Accumulator Final Accumulator Accel
   p27r03_winder_b_distance : REAL := 12.3;
   p27r04 : routine := (comment := -1073741761);   // Winder Output
        .UNACK_FAULT   // Lower Poly Letoff Output Unacknoledged Fault Exist
        .UNACK_WARNING   // Lower Poly Letoff Outputs Unacknoledged Warnnings Exist
   p27r04_timer_fault : TIMER[4];   // Winder Output Fault Delay
   p27r04_timer_warning : TIMER[4];   // Winder Output Warning Delay
   p27r05 : routine := (comment := -1073741761);   // Winder Dint to HMI
        .UNACK_FAULT   // Lower Poly Letoff Dint to HMI Unacknoledged Fault Exist
        .UNACK_WARNING   // Lower Poly Letoff Dint to HMI Unacknoledged Warnnings Exist
   p27r05_lla_mode_tension : BOOL;   // Lower Poly Letoff Modes A Tension Mode
   p27r05_llb_mode_tension : BOOL;   // Lower Poly Letoff Modes B Tension Mode
   p27r05_timer_fault : TIMER[4];   // Winder Dint to HMI Fault Delay
   p27r05_timer_warning : TIMER[4];   // Winder Dint to HMI Warning Delay
   p27r06 : routine := (comment := -1073741572);   // Winder Real to HMI
        .UNACK_FAULT   // Lower Poly Letoff Real to HMI Unacknoledged Fault Exist
        .UNACK_WARNING   // Lower Poly Letoff Real to HMI Unacknoledged Warnnings Exist
   p27r06_timer_fault : TIMER[4];   // Winder Real to HMI Fault Delay
   p27r06_timer_warning : TIMER[4];   // Winder Real to HMI Warning Delay
   p27r07 : routine := (comment := -1073741761);   // Winder Alarms
        .UNACK_FAULT   // Lower Poly Letoff Alarms Unacknoledged Fault Exist
        .UNACK_WARNING   // Lower Poly Letoff Alarms Unacknoledged Warnnings Exist
   p27r07_timer_fault : TIMER[4];   // Winder Alarms Fault Delay
   p27r07_timer_warning : TIMER[4];   // Winder Alarms Warning Delay
   p27r08 : routine := (comment := -1073741761);   // Winder Warnings
        .UNACK_FAULT   // Lower Poly Letoff Warnings Unacknoledged Fault Exist
        .UNACK_WARNING   // Lower Poly Letoff Warnings Unacknoledged Warnnings Exist
   p27r08_timer_fault : TIMER[4];   // Winder Warnings Fault Delay
   p27r08_timer_warning : TIMER[4];   // Winder Warnings Warning Delay
   p27r09 : routine := (comment := -1073741761);   // Winder Modes
        .UNACK_FAULT   // Lower Poly Letoff Modes Unacknoledged Fault Exist
        .UNACK_WARNING   // Lower Poly Letoff Modes Unacknoledged Warnnings Exist
   p27r09_a_enable_toggle : SYS_Toggle;   // Lower Poly Letoff Modes A Toggle
   p27r09_b_enable_toggle : SYS_Toggle;   // Lower Poly Letoff Modes B Toggle
   p27r09_timer_fault : TIMER[4];   // Winder Modes Fault Delay
   p27r09_timer_warning : TIMER[4];   // Winder Modes Warning Delay
   p27r10 : routine := (comment := -1073741777);   // Winder Winder Speed
        .FAULT   // Lower Poly Letoff Lower Poly Letoff Speed Faults
        .UNACK_FAULT   // Lower Poly Letoff Speed Unacknoledged Fault Exist
        .UNACK_WARNING   // Lower Poly Letoff Tension Unacknoledged Warnnings Exist
   p27r10_lla_selected_tension : REAL := 2.0;   // Lower Poly Letoff Tension A Selected Tension
   p27r10_llb_selected_tension : REAL := 2.0;   // Lower Poly Letoff Tension B Selected Tension
   p27r10_timer_fault : TIMER[4];   // Winder Fault Delay
   p27r10_timer_warning : TIMER[4];   // Winder Warning Delay
   p27r10_unwind_a_brake_torque : REAL := -1.098723;   // Lower Poly Letoff Tension Letoff A Brake Torque [lb-ft]
   p27r10_unwind_a_dia_ft : REAL := -0.81831867;   // Lower Poly Letoff Tension Diameter A [ft]
   p27r10_unwind_b_brake_torque : REAL := -7.1031704;   // Lower Poly Letoff Tension Letoff B Brake Torque [lb-ft]
   p27r10_unwind_b_dia_ft : REAL := -7.1031704;   // Lower Poly Letoff Tension Diameter B [ft]
   p27r11 : routine;   // Winder Feedroll
        .UNACK_FAULT   // Lower Poly Letoff Feedroll Unacknoledged Fault Exist
   p289_di_ss_jog : BOOL;   // Winder Digital Input SS:Run/Off/Jog Jog
   p289_di_ss_run : BOOL;   // Winder Digital Input SS:Run/Off/Jog Run
   p28_ai_slitter_amps : REAL;
   p28_ai_slitter_hz : REAL := -3.8146973e-06;
   p28_ai_slitter_speed : REAL;
   p28_ai_sltr_speed : REAL;
   p28_ao_sltr_selected_speed : REAL;
   p28_di_brake : BOOL := 1;
   p28_di_motor : BOOL := 1;
   p28_di_slitter : acs800_di_normal := (ready := 1, ctrl_from_net := 1, ref_from_net := 1);
   p28_dint_to_hmi : DINT[16] := ([1] := 1136);
   p28_do_slt_air_supply_sv : BOOL;
   p28_do_sltr : acs800_do_normal;
   p28_real_to_hmi : REAL[112] := ([7] := -3.8146973e-06);
   p28_slitter_on : SYS_Toggle;
   p28r01 : routine := (comment := 7);
   p28r02 : routine := (comment := -1073741761);
   p28r02_fault_exists : BOOL;
   p28r02_timer_fault : TIMER[4];
   p28r02_timer_warning : TIMER[4];
   p28r02_unack_fault : BOOL;
   p28r02_unack_warning : BOOL;
   p28r02_warning_exists : BOOL;
   p28r03 : routine := (comment := -1073741777);
   p28r03_hz : SYS_SCP := (Input_Max := 1800.0, Output_Max := 60.0, Output := -3.8146973e-06);
   p28r03_slitter_speed_fb : SYS_RPM_TO_SPEED := (IN_gear_ratio := 74.24, IN_roll_diameter := 0.5);
   p28r03_timer_fault : TIMER[4];
   p28r03_timer_warning : TIMER[4];
   p28r04 : routine := (comment := -1073741809);
   p28r04_slitter_gear_ratio : REAL := 74.24;
   p28r04_slitter_roll_diameter_ft : REAL := 0.5;
   p28r04_slitter_speed : SYS_SPEED_TO_VFD := (IN_gear_ratio := 74.24, IN_roll_diameter := 0.5);
   p28r04_timer_fault : TIMER[4];
   p28r04_timer_warning : TIMER[4];
   p28r05 : routine := (comment := -1073741809);
   p28r05_timer_fault : TIMER[4];
   p28r05_timer_warning : TIMER[4];
   p28r06 : routine := (comment := -1073741793);
   p28r06_timer_fault : TIMER[4];
   p28r06_timer_warning : TIMER[4];
   p28r07 : routine := (comment := -1073741817);
   p28r07_timer_fault : TIMER[4];
   p28r07_timer_warning : TIMER[4];
   p28r08 : routine := (comment := -1073741769);
   p28r08_timer_fault : TIMER[4];
   p28r08_timer_warning : TIMER[4];
   p28r09 : routine := (comment := -1073741761);
   p28r09_timer_fault : TIMER[4];
   p28r09_timer_warning : TIMER[4];
   p28r10_request_line_run : BOOL;
   p28r11 : routine := (comment := -1073741713);
   p28r11_permissive_run : BOOL := 1;
   p28r11_request_line_jog : BOOL;
   p28r11_request_line_run : BOOL;
   p28r11_request_thread_fwd : BOOL;
   p28r11_request_thread_rev : BOOL;
   p28r11_slitter_on : BOOL;
   p28r11_timer_fault : TIMER[10];
   p28r11_timer_warning : TIMER[5];
   p29_ai_radius : REAL := 36.375;   // Winder Input Winder Roll Radius [in]
   p29_ai_wa_amps : REAL;   // Winder Analog Inputs Winder A Amps
   p29_ai_wa_dia_ft : REAL := 0.27083334;   // Winder Analog Inputs Winder Roll Diameter [ft]
   p29_ai_wa_hz : REAL;   // Winder Analog Inputs Winder A Hertz
   p29_ai_wa_rpm : REAL := -0.1;   // Winder Analog Inputs Winder A RPM
   p29_ai_wa_speed : REAL := -0.0016729205;   // Winder Analog Inputs Winder A Speed
   p29_ai_wa_torque : REAL;   // Letoff Outputs Letoff Alarm With Manual Fill
   p29_ai_wb_amps : REAL;   // Winder Analog Inputs Winder B Amps
   p29_ai_wb_dia_ft : REAL := 0.282082;
   p29_ai_wb_hz : REAL;   // Winder Analog Inputs Winder B Hertz
   p29_ai_wb_rpm : REAL;   // Winder Analog Inputs Winder B RPM
   p29_ai_wb_speed : REAL;   // Winder Analog Inputs Winder B Speed FB
   p29_ai_wb_torque : REAL;   // Letoff Outputs Letoff Alarm with Auto Fill
   p29_ai_wdr_dia_in : REAL;   // Winder Input Winder Roll Diameter [in]
   p29_ai_wdr_lc : REAL := 85.42392;   // Winder Analog Input Winder Load Cell
   p29_ai_wdr_turret_amps : REAL;   // Winder Analog Inputs Winder Turret Amps
   p29_ai_wdr_turret_hz : REAL;   // Winder Analog Inputs Liner Winder Hertz
   p29_ai_wdr_turret_speed : REAL;   // Winder Analog Inputs Winder Turret Speed
   p29_ao_wa_torque_ref : REAL := 15.2807;
   p29_ao_wb_torque_ref : REAL := 15.500027;
   p29_ao_wda_vfd : REAL;
   p29_ao_wdb_vfd : REAL;
   p29_ao_wdr_turret_selected_speed : REAL;   // Winder Winder Turret VFD AO: Selected Speed
   p29_ao_wdra_selected_speed : REAL;   // Winder Winder A VFD AO: Selected Speed
   p29_ao_wdrb_selected_speed : REAL;   // Winder Winder B VFD AO: Selected Speed
   p29_di_turret_pos : BOOL := 1;   // Winder Digital Input PRX: Winder Turret In Position
   p29_di_wa_brake : BOOL := 1;   // Winder Digital Input Winder A VFD Brake Temperature
   p29_di_wa_motor : BOOL;   // Winder Digital Input Winder A VFD Motor Temperature
   p29_di_wb_brake : BOOL := 1;   // Winder Digital Input Winder B VFD Brake Temperature Ok
   p29_di_wb_motor : BOOL := 1;   // Winder Digital Input Winder B VFD Motor Temperature Ok
   p29_di_wdr_a : BOOL := 1;   // Winder Digital Input SS: Winder B Selected
   p29_di_wdr_a_core_size : BOOL;   // Winder Digital Input SS: Winder A Core Size 3" or 6" 6" Selected
   p29_di_wdr_a_reset_core : BOOL;   // Winder Digital Input PB: Winder A Reset Core
   p29_di_wdr_a_start : BOOL;   // Winder Digital Input PB: Winder A START
   p29_di_wdr_a_stop : BOOL;   // Winder Digital Input PB: Winder A STOP
   p29_di_wdr_b_core_size : BOOL;   // Winder Digital Input SS: Winder B Core Size 3" or 6" 6" Selected
   p29_di_wdr_b_reset_core : BOOL;   // Winder Digital Input PB: Winder B Reset Core
   p29_di_wdr_b_start : BOOL;   // Winder Digital Input PB: Winder B START
   p29_di_wdr_b_stop : BOOL;   // Winder Digital Input PB: Winder B STOP
   p29_di_wdr_index_fwd : BOOL;   // Winder Digital Input PB: Winder Turret Index FWD
   p29_di_wdr_jog : BOOL;   // Winder Digital Input PB: JOG
   p29_di_wdr_turret : acs800_di_normal := (ready := 1, ctrl_from_net := 1, ref_from_net := 1);   // Winder Digital Inputs Turret VFD
   p29_di_wt_motor : BOOL := 1;   // Winder Digital Input Winder Turret Motor Temperature Ok [NOT EXISTING]
   p29_dint_to_hmi : DINT[16] := ([0] := 5, [1] := 5939, [3] := 4785, [4] := 536, [5] := 112);   // Winder Dint to HMI
        [0]   // Winder Dint to HMI Alarms
        [0].0   // Winder Dint to HMI Winder A Active
        [0].1   // Winder Dint to HMI Winder B Active
        [0].2   // Winder Dint to HMI Winder Turret in Position
        [1].0   // Winder Dint to HMI Winder A VFD Faulted
        [1].1   // Winder Dint to HMI Winder A VFD Warning
        [1].2   // Winder Dint to HMI Winder A VFD Running Forward
        [1].3   // Winder Dint to HMI Winder A VFD Running Reverse
        [1].4   // Winder Dint to HMI Winder A VFD Ready
        [1].5   // Winder Dint to HMI Winder A VFD Control from Net
        [1].6   // Winder Dint to HMI Winder A VFD Referecne from Net
        [1].7   // Winder Dint to HMI Winder A VFD At Reference
        [2].0   // Winder Alarms A00: Winder A VFD Faulted
        [2].1   // Winder Alarms A01:
        [2].2   // Winder Alarms A02: Winder A VFD Drive Not Ready
        [2].3   // Winder Alarms A03: Winder A VFD Drive Not in Remote Mode
        [2].4   // Winder Alarms A04: Winder A Motor Temperature
        [2].5   // Winder Alarms A05: Winder A Brake Temperature
        [2].6   // Winder Alarms A06: Winder A High Tension Fault
        [2].7   // Winder Alarms A07:
        [2].8   // Winder Alarms A08: Winder B VFD Faulted
        [2].9   // Winder Alarms A09:
        [2].10   // Winder Alarms A10: Winder B VFD Drive Not Ready
        [2].11   // Winder Alarms A11: Winder B VFD Drive Not in Remote Mode
        [2].12   // Winder Alarms A12: Winder B Motor Temperature
        [2].13   // Winder Alarms A13: Winder B Brake Temperature
        [2].14   // Winder Alarms A14: Winder B High Tension Fault
        [2].15   // Winder Alarms A15:
        [2].16   // Winder Alarms A16: Winder Turret VFD Drive Faulted
        [2].17   // Winder Alarms A17:
        [2].18   // Winder Alarms A18: Winder Turret VFD Drive Not Ready
        [2].19   // Winder Alarms A19: Winder Turret VFD Not in Remote Mode
        [2].20   // Winder Alarms A20: Winder Turret Motor Temperature
        [2].21   // Winder Alarms A21:
        [2].22   // Winder Alarms A22:
        [2].23   // Winder Alarms A23:
        [2].24   // Winder Alarms A24:
        [2].25   // Winder Alarms A25:
        [2].26   // Winder Alarms A26:
        [2].27   // Winder Alarms A27:
        [2].28   // Winder Alarms A28:
        [2].29   // Winder Alarms A29:
        [2].30   // Winder Alarms A30:
        [2].31   // Winder Alarms A31:
        [3].0   // Winder Dint to HMI Winder B VFD Faulted
        [3].1   // Winder Dint to HMI Winder B VFD Warning
        [3].2   // Winder Dint to HMI Winder B VFD Running Forward
        [3].3   // Winder Dint to HMI Winder B VFD Running Reverse
        [3].4   // Winder Dint to HMI Winder B VFD Ready
        [3].5   // Winder Dint to HMI Winder B VFD Control from Net
        [3].6   // Winder Dint to HMI Winder B VFD Reference from Net
        [3].7   // Winder Dint to HMI Winder B VFD At Reference
        [4].0   // Winder Warning W00: Winder A VFD Drive Warning
        [4].1   // Winder Warning W01: Tension Low Deviation
        [4].2   // Winder Warning W02: Tension High Deviation
        [4].3   // Winder Warning W03: Turret Not in Winder A Run Position
        [4].4   // Winder Warning W04: Winder B VFD Drive Warning
        [4].5   // Winder Warning W05: Winder B Tension Low Deviation
        [4].6   // Winder Warning W06: Winder B Tension High Deviation
        [4].7   // Winder Warning W07: Turret Not in Winder B Run Position
        [4].8   // Winder Warning W08: Winder Turret VFD Drive Warning
        [4].9   // Winder Warning W09: No Winder Selected
        [4].10   // Winder Warning W10:
        [4].11   // Winder Warning W11:
        [4].12   // Winder Warning W12:
        [4].13   // Winder Warning W13:
        [4].14   // Winder Warning W14:
        [4].15   // Winder Warning W15:
        [4].16   // Winder Warning W16:
        [4].17   // Winder Warning W17:
        [4].18   // Winder Warning W18:
        [4].19   // Winder Warning W19:
        [4].20   // Winder Warning W20:
        [4].21   // Winder Warning W21:
        [4].22   // Winder Warning W22:
        [4].23   // Winder Warning W23:
        [4].24   // Winder Warning W24:
        [4].25   // Winder Warning W25:
        [4].26   // Winder Warning W26:
        [4].27   // Winder Warning W27:
        [4].28   // Winder Warning W28:
        [4].29   // Winder Warning W29:
        [4].30   // Winder Warning W30:
        [4].31   // Winder Warning W31:
        [5].0   // Winder Dint to HMI Winder Turret VFD Faulted
        [5].1   // Winder Dint to HMI Winder Turret VFD Warning
        [5].2   // Winder Dint to HMI Winder Turret VFD Running Forward
        [5].3   // Winder Dint to HMI Winder Turret VFD Running Reverse
        [5].4   // Winder Dint to HMI Winder Turret VFD Ready
        [5].5   // Winder Dint to HMI Winder Turret VFD Control from Net
        [5].6   // Winder Dint to HMI Winder Turret VFD Reference from Net
        [5].7   // Winder Dint to HMI Winder Turret VFD At Reference
        [13].0   // Laminator Dint to HMI PI: Laminator Drive Fault
        [13].1   // Laminator Dint to HMI PI: Laminator Drive Warning
        [13].2   // Laminator Dint to HMI PI: Laminator Drive Running Forward
        [13].3   // Laminator Dint to HMI PI: Laminator Drive Running Reverse
        [13].4   // Laminator Dint to HMI PI: Laminator Drive Ready
        [13].5   // Laminator Dint to HMI PI: Laminator Drive Control from Net
        [13].6   // Laminator Dint to HMI PI: Laminator Drive Reference from Net
        [13].7   // Laminator Dint to HMI PI: Laminator Drive At Reference
   p29_do_wdr_turret : acs800_do_normal;   // Winder Digital Outpus Winder Turret VFD
   p29_param_acc_park_sp : REAL := 5.0;   // Winder Accumulator Speed Trim Park Setpoint - Where the Carriage Sits [% of Stroke]
   p29_param_acc_trim_gain : REAL := 0.02;   // Winder Accumulator Speed Trim Proportional Gain Fraction of Line Speed per % of Stroke
   p29_param_acc_trim_gain_lo : REAL := 0.05;   // Winder Accumulator Speed Trim Proportional Gain BELOW Park Fraction of Line Speed per % of Stroke Higher than the above-park gain - only 10% of stroke to work with
   p29_param_fast_turret_speed : REAL := 7.0;
   p29_param_index_trim_fpm : REAL := 12.0;   // Winder Accumulator Speed Trim Index Authority - ABSOLUTE fpm Applied both ways during a turret index Size to turret rate x swing radius
   p29_param_lc_cal_factor : REAL := 1.0;   // Winder Load Cell Calibration Factor Applied After Scaling 1.0 - the span is now correct in the scaling itself Was 1.34, trimmed against the old load cell Trim on a known weight if needed
   p29_param_payout_torque : REAL := 100.0;   // Winder Torque Limit During Accumulator Payout Line Running [%]
   p29_param_slow_turret_speed : REAL := 5.0;
   p29_param_soak : REAL := 25.0;
   p29_param_speed_trim_max : REAL := 0.5;   // Winder Accumulator Speed Trim Maximum - Fraction of Line Speed 0.20 = 1.20x line speed, the payout overspeed cap Also sets where the taper starts: park + max/gain = 10 + 10 = 20%
   p29_param_speed_trim_min : REAL := -1.0;   // Winder Accumulator Speed Trim Minimum - Fraction of Line Speed -1.00 = winder commanded to a stop No drive limit on the slow side, and reverse is blocked downstream
   p29_param_start_speed_factor : REAL := 0.5;   // Winder Start Speed Fraction of Line Speed Before Tension is Established Shared by Winder A and B
   p29_param_tension_ok_band : REAL := 15.0;   // Winder Tension Established Band Shared by Winder A and B [lbf]
   p29_param_turret_encoder_enable : BOOL;   // Winder Parameter Turret Encoder Enable 0 = original prox index (commissioning default) 1 = encoder positioning
   p29_param_wa_gear_ratio : REAL := 50.86;   // Winder Parameter Winder A Gear Ratio
   p29_param_wb_gear_ratio : REAL := 50.86;   // Winder Parameter Winder B Gear Ratio
   p29_param_wdt_gear_ratio : REAL := 1200.0;
   p29_param_wind_out_speed : REAL := 5.0;   // Winder Wind Out Speed Winder Speed with the Line Stopped Empties the Accumulator [fpm]
   p29_param_wind_out_stop_pct : REAL := 5.0;   // Winder Wind Out Stop When the Accumulator Reaches This Position [% of Stroke]
   p29_param_wind_out_torque : REAL := 50.0;   // Winder Torque Limit During Wind Out Line Stopped [%]
   p29_param_winder_accel_rate : REAL := 25.0;   // Winder Common Speed Ramp Default Accel Rate Applied Only if winder_accel_rate is Zero
   p29_param_winder_decel_rate : REAL := 25.0;   // Winder Common Speed Ramp Default Decel Rate Applied Only if winder_decel_rate is Zero
   p29_param_winder_jog_speed : REAL := 8.0;   // System Parameters Winder Jog Speed
   p29_real_to_hmi : REAL[112] := ([1] := 85.40576, [3] := 3.25, [4] := 3.384984, [6] := -0.0016729205, [21] := 49.682617, [22] := 723.2029, [40] := 2.5, [41] := 0.9);   // Laminator Real to HMI
        [0]   // Laminator Real to HMI
   p29_wa_footage_input_max : REAL := 9000.0;
   p29_wa_footage_input_min : REAL;
   p29_wa_footage_output_max : REAL := 9000.0;
   p29_wa_footage_output_min : REAL;
   p29_wb_footage_input_max : REAL := 9000.0;
   p29_wb_footage_input_min : REAL;
   p29_wb_footage_output_max : REAL := 9000.0;
   p29_wb_footage_output_min : REAL;
   p29_wda_control_word : INT := 2#0000_0100_0000_0111;
   p29_wda_status_word : INT := 2#0001_0111_0011_0011;
   p29_wda_vfd : ABB_PROTOCOL_VFD := (STATUS_WORD := 5939, CONTROL_WORD := 1031, IN_DRIVE_PERMISSIVE := 1);
   p29_wda_vfd_input_max : REAL := 2000.0;
   p29_wda_vfd_input_min : REAL := -2000.0;
   p29_wda_vfd_output_max : REAL := 20000.0;
   p29_wda_vfd_output_min : REAL := -20000.0;
   p29_wdb_control_word : INT := 2#0000_0100_0000_0110;
   p29_wdb_status_word : INT := 2#0001_0010_1011_0001;
   p29_wdb_vfd : sys_ACS_FENA21 := (IN_DRIVE_PERMISSIVE := 1, OUT_ALARM := 1);
   p29_wdb_vfd_input_max : REAL := 2000.0;
   p29_wdb_vfd_input_min : REAL := -2000.0;
   p29_wdb_vfd_output_max : REAL := 20000.0;
   p29_wdb_vfd_output_min : REAL := -20000.0;
   p29_wdr_diameter_input_max : REAL := 30959.0;
   p29_wdr_diameter_input_min : REAL := 100.0;
   p29_wdr_diameter_output_max : REAL := 55.0;
   p29_wdr_diameter_output_min : REAL := 4.0;
   p29_wdr_lc_input_max : REAL := 20000.0;   // Winder Load Cell Scaling Input Maximum 20 mA on p00_io_winder:2:I.Ch6Data Was 10000 for the old Local:3:I.Ch2 card - that clamped the reading above 10 mA
   p29_wdr_lc_input_min : REAL := 4000.0;   // Winder Load Cell Scaling Input Minimum 4 mA on p00_io_winder:2:I.Ch6Data Accumulator exit load cell
   p29_wdr_lc_output_max : REAL := 200.0;   // Winder Load Cell Scaling Output Maximum Load cell calibrated full scale Matches the P31 ai_ten01 scaling on the same channel [lbf]
   p29_wdr_lc_output_min : REAL;   // Winder Load Cell Scaling Output Minimum [lbf]
   p29_winder_at_run_position : BOOL;   // Winder Payout Interlock Selected winder is at ITS OWN turret run position Controller scope - p31 cannot see the p29 position bits
   p29r01 : routine := (comment := 7);
   p29r02 : routine := (comment := -1073741761);
        .UNACK_FAULT   // Winder Misc Control Unacknowleged Faults Exist
        .UNACK_WARNING   // Winder Misc Control Unacknowleged Warnings Exist
   p29r02_fault_exists : BOOL;
   P29r02_pb_roll_count_reset : BOOL;   // Production Roll Count Reset
   P29r02_roll_count : DINT;   // Production Roll Count
   p29r02_tension_dev_max : REAL := 76.0;
   p29r02_tension_dev_min : REAL := 64.0;
   p29r02_timer_fault : TIMER[4];   // Winder Misc Control Fault Dwell Timer
   p29r02_timer_warning : TIMER[4];   // Winder Misc Control Warning Dwell Timer
   p29r02_unack_fault : BOOL;   // Winder Misc Control Unacknowledged Fault Exists
   p29r02_unack_warning : BOOL := 1;   // Winder Misc Control Unackn. Warning Exists
   p29r02_wa_calc_torque_ref : REAL := 108.33333;   // Zone 2 Digital Input Recirculation Air Filter Dirty
   p29r02_warning_exists : BOOL := 1;
   p29r02_wb_calc_torque_ref : REAL := 112.832794;
   p29r02_winder_selection_dwell : TIMER := (PRE := 60000, EN := 1, DN := 1);
   p29r03 : routine := (comment := -1073741761);
        .UNACK_FAULT   // Winder Input Unacknowleged Faults Exist
        .UNACK_WARNING   // Winder Input Unacknowleged Warnings Exist
   p29r03_distance_to_core : REAL := 40.375;
   p29r03_hz : SYS_SCP := (Input_Max := 2000.0, Output_Max := 60.0);   // Winder Analog Inputs SCP Hz
   p29r03_liner_wdr_lc_scp : SYS_SCP := (Input := 10811.0, Input_Min := 4000.0, Input_Max := 20000.0, Output_Max := 200.0, Output := 85.1375);   // Winder Analog Input Winder Load Cell
   p29r03_sample_timer : TIMER := (PRE := 200, ACC := 33, EN := 1, TT := 1);
   p29r03_sensor_input : REAL := 4.0;
   p29r03_timer_fault : TIMER[4];   // Winder Input Fault Dwell Timer
   p29r03_timer_warning : TIMER[4];   // Winder Input Warning Dwell Timer
   p29r03_unload : REAL;
   p29r03_wa_ave_tq : REAL;
   p29r03_wa_footage_scp : SYS_SCP := (Input := 49.541016, Input_Max := 9000.0, Output_Max := 9000.0, Output := 49.541016);   // Winder Analog Inputs Winder A Footage Counter Scaling
   p29r03_wa_scaled_vfd_in : REAL := -0.1;
   p29r03_wa_speed_fb : SYS_RPM_TO_SPEED := (IN_gear_ratio := 50.86, IN_roll_diameter := 0.27083334, IN_vfd_fb_rpm := -0.1, OUT_surface_speed_fb := -0.0016729205);   // Winder Analog Inputs Winder A Speed FB
   p29r03_wa_tq_ave_ctrl : CONTROL := (LEN := 19);   // Letoff Outputs Letoff Alarm LMMI
   p29r03_wa_tq_buffer : REAL[20];
   p29r03_wa_tq_fifo : CONTROL := (LEN := 20, POS := 20, DN := 1);
   p29r03_wb_ave_tq : REAL;   // Impreg Metering Roll VFD Mean +
   p29r03_wb_footage_scp : SYS_SCP := (Input := 722.92017, Input_Max := 9000.0, Output_Max := 9000.0, Output := 722.92017);   // Winder Analog Inputs Winder B Footage Counter Scaling
   p29r03_wb_scaled_vfd_in : REAL;
   p29r03_wb_speed_fb : SYS_RPM_TO_SPEED := (IN_gear_ratio := 50.86, IN_roll_diameter := 0.27083334);   // Winder Analog Inputs Winder B Speed FB
   p29r03_wb_tq_ave_ctrl : CONTROL := (LEN := 19);
   p29r03_wb_tq_buffer : REAL[20];   // Impreg Metering Roll VFD Mean -
   p29r03_wb_tq_fifo : CONTROL := (LEN := 20, POS := 20, DN := 1);
   p29r03_wda_vfd_in_scaling : SYS_SCP := (Input := -1.0, Input_Min := -20000.0, Input_Max := 20000.0, Output_Min := -2000.0, Output_Max := 2000.0, Output := -0.1);
   p29r03_wda_vfd_input_max : REAL := 20000.0;
   p29r03_wda_vfd_input_min : REAL := -20000.0;
   p29r03_wda_vfd_output_max : REAL := 2000.0;
   p29r03_wda_vfd_output_min : REAL := -2000.0;
   p29r03_wdb_vfd_in_scaling : SYS_SCP := (Input_Min := -20000.0, Input_Max := 20000.0, Output_Min := -2000.0, Output_Max := 2000.0);
   p29r03_wdb_vfd_input_max : REAL := 20000.0;
   p29r03_wdb_vfd_input_min : REAL := -20000.0;
   p29r03_wdb_vfd_output_max : REAL := 2000.0;
   p29r03_wdb_vfd_output_min : REAL := -2000.0;
   p29r03_wdr_dia_sensor_scp : SYS_SCP := (Input_Min := 100.0, Input_Max := 30959.0, Output_Min := 4.0, Output_Max := 55.0, Output := 4.0);   // Winder Analog Input Winder Roll Diameter Sensor Scaling
   p29r04 : routine := (comment := -1073741761);
        .UNACK_FAULT   // Winder Output Unacknowleged Faults Exist
        .UNACK_WARNING   // Winder Output Unacknowleged Warnings Exist
   p29r04_timer_fault : TIMER[4];   // Winder Output Fault Dwell Timer
   p29r04_timer_warning : TIMER[4];   // Winder Output Warning Dwell Timer
   p29r04_wda_vfd_out_scaling : SYS_SCP := (Input_Min := -2000.0, Input_Max := 2000.0, Output_Min := -20000.0, Output_Max := 20000.0);
   p29r04_wdb_vfd_out_scaling : SYS_SCP := (Input_Min := -2000.0, Input_Max := 2000.0, Output_Min := -20000.0, Output_Max := 20000.0);
   p29r04_wdr_turret_speed_to_vfd : SYS_SPEED_TO_VFD := (IN_gear_ratio := 1200.0, IN_roll_diameter := 3.2);
   p29r04_wdra_speed_to_vfd : SYS_SPEED_TO_VFD := (IN_gear_ratio := 50.86, IN_roll_diameter := 0.27083334);   // Winder Analog Outputs Winder A Speed
   p29r04_wdrb_speed_to_vfd : SYS_SPEED_TO_VFD := (IN_gear_ratio := 50.86, IN_roll_diameter := 0.27083334);   // Winder Analog Outputs Winder B Speed
   p29r05 : routine := (comment := -1073741761);
        .UNACK_FAULT   // Winder Dint to HMI Unacknowleged Faults Exist
        .UNACK_WARNING   // Winder Dint to HMI Unacknowleged Warnings Exist
   p29r05_timer_fault : TIMER[4];   // Winder Dint to HMI Fault Dwell Timer
   p29r05_timer_warning : TIMER[4];   // Winder Dint to HMI Warning Dwell Timer
   p29r06 : routine := (comment := -1073741572);
        .UNACK_FAULT   // Winder Real to HMI Unacknowleged Faults Exist
        .UNACK_WARNING   // Winder Real to HMI Unacknowleged Warnings Exist
   p29r06_ave_wdr_lc : REAL := 85.412865;
   p29r06_lc_buffer : REAL[20] := ([0] := 85.4093, [1] := 85.42839, [2] := 85.40944, [3] := 85.40848, [4] := 85.407555, [5] := 85.42671, [6] := 85.407326, [7] := 85.40645, [8] := 85.404076, [9] := 85.423935, [10] := 85.4057, [11] := 85.406456, [12] := 85.42416, [13] := 85.4059, [14] := 85.42101, [15] := 85.40342, [16] := 85.40428, [17] := 85.385544, [18] := 85.40286, [19] := 85.402176);
   p29r06_sample_timer : TIMER := (PRE := 200, ACC := 165, EN := 1, TT := 1);
   p29r06_timer_fault : TIMER[4];   // Winder Real to HMI Fault Dwell Timer
   p29r06_timer_warning : TIMER[4];   // Winder Real to HMI Warning Dwell Timer
   p29r06_unload : REAL := 85.41028;
   p29r06_wdr_lc_ave_ctrl : CONTROL := (LEN := 19);
   p29r06_wdr_lc_fifo : CONTROL := (LEN := 20, POS := 20, DN := 1);
   p29r07 : routine := (comment := -1073741761);
        .UNACK_FAULT   // Winder Alarms Unacknowleged Faults Exist
        .UNACK_WARNING   // Winder Alarms Unacknowleged Warnings Exist
   p29r07_timer_fault : TIMER[4];   // Winder Alarms Fault Dwell Timer
   p29r07_timer_warning : TIMER[4];   // Winder Alarms Warning Dwell Timer
   p29r08 : routine := (comment := -1073741761);
        .UNACK_FAULT   // Winder Warnings Unacknowleged Faults Exist
        .UNACK_WARNING   // Winder Warnings Unacknowleged Warnings Exist
   p29r08_timer_fault : TIMER[4];   // Winder Warnings Fault Dwell Timer
   p29r08_timer_warning : TIMER[4];   // Winder Warnings Warning Dwell Timer
   p29r09 : routine := (comment := -1073741761);
        .UNACK_FAULT   // Winder Modes Unacknowleged Faults Exist
        .UNACK_WARNING   // Winder Modes Unacknowleged Warnings Exist
   p29r09_mode_doff_auto : BOOL;   // Winder Mode Doff Position - AUTO Winder A/B doff PB indexes the turret to the preset doff position
   p29r09_mode_doff_manual : BOOL := 1;   // Winder Mode Doff Position - MANUAL Operator jogs the turret to doff, doff PBs do nothing
   p29r09_ten_ave_len : DINT := 19;
   p29r09_ten_len : DINT := 20;
   p29r09_ten_pos : DINT := 19;
   p29r09_tension_mode : BOOL := 1;
   p29r09_timer_fault : TIMER[4];   // Winder Modes Fault Dwell Timer
   p29r09_timer_warning : TIMER[4];   // Winder Modes Warning Dwell Timer
   p29r09_torque_mode : BOOL;
   p29r09_trq_ave_len : DINT := 999;
   p29r09_trq_len : DINT := 1000;
   p29r09_trq_pos : DINT := 999;
   p29r09_winder_a_active : BOOL := 1;   // Winder Modes Winder A Active
   p29r09_winder_b_active : BOOL;   // Winder Modes Winder B Active
   p29r09_winder_jog : BOOL;   // Winder Modes Jog
   p29r09_winder_off : BOOL := 1;   // Winder Modes Off
   p29r09_winder_run : BOOL;   // Winder Modes Run
   p29r10 : routine := (comment := -1073740737, oneshot := 2);
        .UNACK_FAULT   // Winder Winder A Speed Control Unacknowleged Faults Exist
        .UNACK_WARNING   // Winder Winder Speed Control Unacknowleged Warnings Exist
   p29r10_acc_pstn_error : REAL := -5.0853424;   // Winder Winder A Accumulator Position Error position - park setpoint [% of Stroke]
   p29r10_accel_bias : REAL := 1.0;
   p29r10_calc_speed_offset : REAL := -0.0016729205;
   p29r10_index_active : BOOL;   // Winder Winder A VDF Index Active
   p29r10_line_guard : REAL := 1.0;   // Winder Accumulator Speed Trim Line speed, floored at 1.0 fpm for the divide
   p29r10_misc_index_factor : REAL := 70.0;   // Winder Winder A Speed Control Index Factor
   p29r10_param_psn_gain : REAL := 80.0;   // Winder Winder Speed Parameter Gain
   p29r10_pid_out : REAL := 49.99998;
   p29r10_pid_psn : PID := (CTL := -2078243712, EN := 1, SWM := 1, NOBC := 1, INI := 1, DVNA := 1, PVHA := 1, SP := 70.0, KP := 2.5, KI := 0.9, MAXS := 500.0, SO := 49.99998, MAXO := 100.0, UPD := 0.01, PV := 85.352264, ERR := -15.352264, OUT := 49.99998, MAXI := 500.0, MAXCV := 100.0, MAXTIE := 100.0, DATA[0] := 57.676113, DATA[1] := -273.12726, DATA[2] := 85.352264, DATA[3] := -15.352264, DATA[4] := 70.0, DATA[5] := 0.2, DATA[6] := 1.0, DATA[7] := 0.16, DATA[8] := 2.5, DATA[9] := 0.9, DATA[11] := 2.5, DATA[12] := 0.9, DATA[15] := 1.0, DATA[16] := 1.0);   // Winder Winder A Speed Control PID Control
        .SP   // Winder Winder A Speed Control PID
        .SO   // Winder Winder A Speed Control PID
   p29r10_pid_psn_cv : REAL := 49.99998;
   p29r10_pid_psn_pv : REAL := 85.40455;   // Winder Winder Speed Position Process Variable
   p29r10_pid_torque : REAL;
   p29r10_pid_tq : PID := (CTL := -2078243712, EN := 1, SWM := 1, NOBC := 1, INI := 1, DVNA := 1, PVHA := 1, SP := 70.0, KP := 10.0, KI := 0.01, MAXS := 500.0, MAXO := 100.0, UPD := 0.01, PV := 85.33197, ERR := -15.33197, MAXI := 500.0, MAXCV := 80.0, MINCV := 5.0, MAXTIE := 4095.0, DATA[0] := 30.66394, DATA[1] := -273.06232, DATA[2] := 85.33197, DATA[3] := -15.33197, DATA[4] := 70.0, DATA[5] := 0.2, DATA[6] := 1.0, DATA[7] := 0.16, DATA[8] := 10.0, DATA[9] := 0.01, DATA[11] := 10.0, DATA[12] := 0.01, DATA[15] := 0.75, DATA[16] := 0.024420025);   // Winder A PID Torque
   p29r10_pid_tq_cv : REAL := 5.0;
   p29r10_psn_gain : REAL := 80.0;   // Winder Winder A Speed Control Gain
   p29r10_request_run : BOOL;   // Winder Winder A Speed Control Request Run
   p29r10_run_permissive : BOOL := 1;   // Winder Winder A Speed Control Run Permissive
   p29r10_speed_offset : REAL := -2.3841858e-07;
   p29r10_tension_error : REAL := -15.40509;   // Winder Winder A Tension Error winder_tension_sp - Load Cell [lbf]
   p29r10_timer : TIMER[4] := ([0].PRE := 100, [0].ACC := 34, [0].EN := 1, [0].DN := 1);   // Winder Winder Speed Timer
        [0]   // Winder Winder A Speed Control PID Enable Timer
   p29r10_timer_fault : TIMER[4];   // Winder Winder A Speed Control Fault Dwell Timer
   p29r10_timer_warning : TIMER[4];   // Winder Winder A Speed Control Warning Dwell Timer
   p29r10_trim_clamp : sys_Limit_Clamp := (max := 0.2, min := -1.0);   // Winder Winder A Speed Trim Clamp
   p29r10_trim_hi : REAL := 0.2;   // Winder Accumulator Speed Trim Upper limit in use this scan
   p29r10_trim_lo : REAL := -1.0;   // Winder Accumulator Speed Trim Lower limit in use this scan
   p29r11 : routine := (comment := -1073740737);
   p29r11_acc_pstn_error : REAL := -5.0853424;   // Winder Winder B Accumulator Position Error position - park setpoint [% of Stroke]
   p29r11_accel_bias : REAL := 1.0;
   p29r11_calc_speed_offset : REAL;
   p29r11_index_active : BOOL;   // Winder Winder B VFD Index Active
   p29r11_line_guard : REAL := 1.0;   // Winder Accumulator Speed Trim Line speed, floored at 1.0 fpm for the divide
   p29r11_line_start : BOOL;
   p29r11_line_stop : BOOL;
   p29r11_misc_index_factor : REAL := 70.0;   // Winder Winder B Speed Control Index Factor
   p29r11_param_psn_gain : REAL := 80.0;   // Winder Winder B Speed Control PID Gain
   p29r11_pid_out : REAL := 50.0;
   p29r11_pid_psn : PID := (CTL := -2078243712, EN := 1, SWM := 1, NOBC := 1, INI := 1, DVNA := 1, PVHA := 1, SP := 70.0, KP := 2.5, KI := 0.9, MAXS := 300.0, SO := 50.0, MAXO := 100.0, UPD := 0.01, PV := 85.347786, ERR := -15.347786, OUT := 50.0, MAXI := 300.0, MAXCV := 100.0, MAXTIE := 100.0, DATA[0] := 62.78982, DATA[1] := -455.1882, DATA[2] := 85.347786, DATA[3] := -15.347786, DATA[4] := 70.0, DATA[5] := 0.33333334, DATA[6] := 1.0, DATA[7] := 0.16, DATA[8] := 2.5, DATA[9] := 0.9, DATA[11] := 2.5, DATA[12] := 0.9, DATA[15] := 1.0, DATA[16] := 1.0);   // Winder Winder B Speed Control PID
   p29r11_pid_psn_cv : REAL := 50.0;   // Winder Winder B Speed Control PID Control Value
   p29r11_pid_psn_pv : REAL := 85.40518;   // Winder Winder B Speed Control PID PV
   p29r11_pid_torque : REAL;
   p29r11_pid_tq : PID := (CTL := -2080340864, EN := 1, SWM := 1, INI := 1, DVNA := 1, PVHA := 1, SP := 70.0, KP := 10.0, KI := 0.01, MAXS := 4095.0, MAXO := 100.0, UPD := 0.01, PV := 85.402054, ERR := -15.402054, MAXI := 4095.0, MAXTIE := 4095.0, DATA[0] := 3.7611854, DATA[1] := -33.368324, DATA[2] := 85.402054, DATA[3] := -15.402054, DATA[4] := 70.0, DATA[5] := 0.024420025, DATA[6] := 1.0, DATA[7] := 0.16, DATA[8] := 10.0, DATA[9] := 0.01, DATA[11] := 10.0, DATA[12] := 0.01, DATA[16] := 0.024420025);   // Winder B PID Torque
   p29r11_pid_tq_cv : REAL;   // Tension Stand 2 VFD
        .DATA[0]   // Input Tension Stand 2 VFD Status Word
        .DATA[0].0   // Input Tension Stand 2 VFD Faulted
        .DATA[0].1   // Input Tension Stand 2 VFD Warning
        .DATA[0].2   // Input Tension Stand 2 VFD Running Forward
        .DATA[0].3   // Input Tension Stand 2 VFD Running Reverse
        .DATA[0].4   // Input Tension Stand 2 VFD Ready
        .DATA[0].5   // Input Tension Stand 2 VFD Control from Net
        .DATA[0].6   // Input Tension Stand 2 VFD Reference from Net
        .DATA[0].7   // Input Tension Stand 2 VFD At Reference
        .DATA[1]   // Input Tension Stand 2 VFD Speed
        .DATA[2]   // Input Tension Stand 2 VFD Amps
        .DATA[3]   // Input Tension Stand 2 VFD Max Hertz
        .DATA[4]   // Input Tension Stand 2 VFD Motor Nameplate Hertz
        .DATA[5]   // Input Tension Stand 2 VFD Motor Nameplate RPM
   p29r11_psn_gain : REAL := 80.0;   // Winder Winder B Speed Control PID Gain
   p29r11_request_run : BOOL;   // Winder Winder B Speed Control Request Run
   p29r11_run_permissive : BOOL := 1;   // Winder Winder B Speed Control Run Permissive
   p29r11_speed_offset : REAL;
   p29r11_tension_error : REAL := -15.403992;   // Winder Winder B Tension Error winder_tension_sp - Load Cell [lbf]
   p29r11_timer : TIMER[1] := ([0].PRE := 100, [0].ACC := 133, [0].EN := 1, [0].DN := 1);   // Winder Winder B Speed Control PID Enable Timer
   p29r11_timer_fault : TIMER[4];   // Winder Winder B Speed Control Fault Dwell Timer
   p29r11_timer_warning : TIMER[4];   // Winder Winder B Speed Control Warning Dwell Timer
   p29r11_trim_clamp : sys_Limit_Clamp := (max := 0.2, min := -1.0);   // Winder Winder B Speed Trim Clamp
   p29r11_trim_hi : REAL := 0.2;   // Winder Accumulator Speed Trim Upper limit in use this scan
   p29r11_trim_lo : REAL := -1.0;   // Winder Accumulator Speed Trim Lower limit in use this scan
   p29r13_ai_wa_footage_ft : REAL := 49.541016;
   p29r13_ai_wb_footage_ft : REAL := 722.92017;
   p29r15 : routine := (comment := -1073741577, warning := 8, unack_warning := 1);   // Winder Winder A VFD
        .FAULT.0   // Winder Winder A VFD Drive Fault
        .FAULT.2   // Winder Winder A VFD Drive Not Ready
        .FAULT.3   // Winder Winder A VFD Drive No In Remote Mode
        .FAULT.4   // Winder Winder A VFD Motor Temperature
        .FAULT.5   // Winder Winder A VFD Brake Temperature
        .FAULT.6   // Winder Winder A VFD High Tension Fault
        .WARNING.0   // Winder Winder A VFD Drive Warning
        .WARNING.1   // Winder Winder A VFD Tension Low Deviation
        .WARNING.2   // Winder Winder A VFD Tension High Deviation
        .WARNING.3   // Winder Winder A VFD Turret Not in Winder A Run Position
        .UNACK_FAULT   // Winder Winder A VFD Unacknowleged Faults Exist
        .UNACK_WARNING   // Winder Winder A VFD Unacknowleged Warnings Exist
   p29r15_accel_rate : REAL := 25.0;   // Winder Winder A VFD Accel Rate
   p29r15_acel_decel_ramp : SYS_ACC_DEC_RAMP := (IN_param_master_accel_rate := 25.0, IN_param_master_decel_rate := 25.0, IN_last_scan_s := 0.032284);   // Winder A Speed Setpoint Ramp
   p29r15_ao_torque : REAL := 28.89195;
   p29r15_const_torque_ref : REAL := 36.0;
   p29r15_decel_rate : REAL := 25.0;   // Winder Winder A VFD Decel Rate
   p29r15_fast_accel_rate : REAL := 25.0;
   p29r15_fast_decel_rate : REAL := 25.0;
   p29r15_index_start_torque : REAL;
   p29r15_jog_torque_ref : REAL := 100.0;
   p29r15_ramped_setpoint : REAL;   // Winder A Ramped Speed Setpoint [fpm]
   p29r15_request_jog_fwd : BOOL;   // Winder Winder A VFD Request Jog FWD
   p29r15_request_run : BOOL;   // Winder Winder A VFD Request Run
   p29r15_request_thread_fwd : BOOL;
   p29r15_request_thread_rev : BOOL;
   p29r15_run_permissive : BOOL := 1;   // Winder Winder A VFD Permissive Run
   p29r15_selected_speed : REAL;   // Winder Winder A VFD Selected Speed
   p29r15_selected_torque : REAL;   // System Annunciators Unacknowledged Fault Exists
   p29r15_soak_active : BOOL := 1;
   p29r15_speed_factor : REAL;   // Winder A Speed Factor Multiplier on the Ramped Setpoint
   p29r15_speed_setpoint : REAL;   // Winder A Speed Setpoint [fpm]
   p29r15_state : DINT := 3;   // Winder Winder A VFD Tension Mode Start Sequence State Word
        .0   // Winder A Sequence Step Gate One Step per Scan
        .1   // Winder A Sequence State 1 Idle / Reset
        .2   // Winder A Sequence State 2 Start - Constant Torque const_torque_ref, Speed Limit 1.5x
        .3   // Winder A Sequence State 3 Tension High torque_low_ref
        .4   // Winder A Sequence State 4 Tension Low torque_high_ref
        .5   // Winder A Sequence State 5 Tension OK
        .6   // Winder A Sequence State 6 Run Enables p29r10_request_run
        .7   // Winder A Sequence State 7 Stopping Returns to State 1
   p29r15_stop_dwell : TIMER := (PRE := 1500, ACC := 1520);   // Winder A Stop Dwell Holds the winder after the stop PB so the nip closes first
   p29r15_tension_ok : BOOL;   // Impreg Supply VFD PID Process Value
   p29r15_thread_torque_ref : REAL := 100.0;   // Letoff A VFD
        .DATA[0]   // Output Letoff A VFD Control Word
        .DATA[0].0   // Output Letoff A VFD Run Forward
        .DATA[0].1   // Output Letoff A VFD Run Reverse
        .DATA[0].2   // Output Letoff A VFD Fault Reset
        .DATA[0].5   // Output Letoff A VFD Net Control
        .DATA[0].6   // Output Letoff A VFD Net Reference
        .DATA[1]   // Output Letoff A VFD Speed Command
   p29r15_timer_fault : TIMER[10] := ([6].PRE := 3000);   // Winder Winder A VFD Fault Dwell Timer
   p29r15_timer_warning : TIMER[4] := ([0].PRE := 10000, [1].PRE := 10000, [2].PRE := 10000);   // Winder Winder A VFD Warning Dwell Timer
   p29r15_torque_acc_rate : REAL := 0.05;   // Zone 1 Recirc VFD Fan Stopped Manually - Prevent Auto Start during Cooldown
   p29r15_torque_boost_acc_rate : REAL := 5000.0;
   p29r15_torque_boost_dec_rate : REAL := 2.0;
   p29r15_torque_boost_ref : REAL := 90.0;
   p29r15_torque_boost_timer : TIMER := (PRE := 500);
   p29r15_torque_dec_rate : REAL := 0.05;   // Zone 1 Recirc VFD PB: Auto Stop
   p29r15_torque_fast_acc_rate : REAL := 0.8;
   p29r15_torque_fast_dec_rate : REAL := 1.6;
   p29r15_torque_high_ref : REAL := 100.0;   // System Annunciators Unacknowledged Fault Exists
   p29r15_torque_low_ref : REAL := 1.0;   // Tension Stand 2 Digital Outputs VFD
   p29r15_torque_mode_acc_rate : REAL := 5000.0;
   p29r15_torque_mode_dec_rate : REAL := 4.0;
   p29r15_torque_ramp : SYS_ACC_DEC_RAMP := (IN_param_master_accel_rate := 0.05, IN_param_master_decel_rate := 0.05, IN_last_scan_s := 0.03258);
   p29r15_torque_soak_acc_rate : REAL := 0.05;
   p29r15_torque_soak_dec_rate : REAL := 0.05;
   p29r15_torque_start_timer : TIMER := (PRE := 200);   // Impreg Supply VFD PID Control Value
   p29r15_vfd_start_request : BOOL;
   p29r15_wdra_accel_decel : SYS_ACC_DEC_RAMP := (IN_param_master_accel_rate := 25.0, IN_param_master_decel_rate := 25.0, IN_last_scan_s := 0.032768);   // Winder Winder A VFD Accel Decel Ramp
   p29r15_wdra_active : BOOL := 1;   // Winder Winder A VFD Winder A Active
   p29r15_wdra_ramped_speed : REAL;   // Winder Winder A VFD Ramped Speed
   p29r15_zero_speed : BOOL := 1;   // Winder Winder A VFD At Zero Speed
   p29r16 : routine := (comment := -1073741577, warning := 1, warning_ack := 9, unack_warning := 1);   // Winder Winder B VFD
        .FAULT.0   // Winder Winder B VFD Drive Faulted
        .FAULT.2   // Winder Winder B VFD Drive Not Ready
        .FAULT.3   // Winder Winder B VFD Drive Not in Remote Mode
        .FAULT.4   // Winder Winder B VFD Motor Temperature
        .FAULT.5   // Winder Winder B VFD Brake Temperature
        .FAULT.6   // Winder Winder B VFD High Tension Fault
        .WARNING.0   // Winder Winder B VFD Drive Warning
        .WARNING.1   // Winder Winder B VFD Tension Low Deviation
        .WARNING.2   // Winder Winder B VFD Tension High Deviation
        .WARNING.3   // Winder Winder B VFD Turret Not in Winder B Run Position
        .UNACK_FAULT   // Winder Winder B VFD Unacknowleged Faults Exist
        .UNACK_WARNING   // Winder Winder B VFD Unacknowleged Warnings Exist
   p29r16_accel_rate : REAL := 25.0;   // Winder Winder B VFD Accel Rate
   p29r16_acel_decel_ramp : SYS_ACC_DEC_RAMP := (IN_param_master_accel_rate := 25.0, IN_param_master_decel_rate := 25.0, IN_last_scan_s := 0.032546);   // Winder B Speed Setpoint Ramp
   p29r16_ao_torque : REAL;
   p29r16_const_torque_ref : REAL := 36.0;   // Winder Winder B VFD Request Jog REV
   p29r16_decel_rate : REAL := 25.0;   // Winder Winder B VFD Decel Rate
   p29r16_fast_accel_rate : REAL := 25.0;
   p29r16_fast_decel_rate : REAL := 25.0;
   p29r16_index_start_torque : REAL;
   p29r16_jog_torque_ref : REAL := 100.0;
   p29r16_ramped_setpoint : REAL;   // Winder B Ramped Speed Setpoint [fpm]
   p29r16_request_jog_fwd : BOOL;   // Winder Winder B VFD Request Jog FWD
   p29r16_request_run : BOOL;   // Winder Winder B VFD Request Run
   p29r16_request_thread_fwd : BOOL;   // Winder Winder B VDF Request Thread Forward
   p29r16_request_thread_rev : BOOL;   // Winder Winder B VDF Request Thread Reverse
   p29r16_run_permissive : BOOL := 1;   // Winder Winder B VFD Run Permissive
   p29r16_selected_speed : REAL;   // Winder Winder B VFD Selected Speed
   p29r16_selected_torque : REAL;
   p29r16_soak_active : BOOL := 1;
   p29r16_speed_factor : REAL;   // Winder B Speed Factor Multiplier on the Ramped Setpoint
   p29r16_speed_setpoint : REAL;   // Winder B Speed Setpoint [fpm]
   p29r16_state : DINT := 3;   // Winder Winder B VFD Tension Mode Start Sequence State Word
        .0   // Winder B Sequence Step Gate One Step per Scan
        .1   // Winder B Sequence State 1 Idle / Reset
        .2   // Winder B Sequence State 2 Start - Constant Torque const_torque_ref, Speed Limit 1.5x
        .3   // Winder B Sequence State 3 Tension High torque_low_ref
        .4   // Winder B Sequence State 4 Tension Low torque_high_ref
        .5   // Winder B Sequence State 5 Tension OK
        .6   // Winder B Sequence State 6 Run Enables p29r11_request_run
        .7   // Winder B Sequence State 7 Stopping Returns to State 1
   p29r16_stop_dwell : TIMER := (PRE := 1500, ACC := 1516);   // Winder B Stop Dwell Holds the winder after the stop PB so the nip closes first
   p29r16_tension_ok : BOOL;
   p29r16_thread_torque_ref : REAL := 100.0;   // Letoff A VFD
        .DATA[0]   // Input Letoff A VFD Status Word
        .DATA[0].0   // Input Letoff A VFD Faulted
        .DATA[0].1   // Input Letoff A VFD Warning
        .DATA[0].2   // Input Letoff A VFD Running Forward
        .DATA[0].3   // Input Letoff A VFD Running Reverse
        .DATA[0].4   // Input Letoff A VFD Ready
        .DATA[0].5   // Input Letoff A VFD Control from Net
        .DATA[0].6   // Input Letoff A VFD Reference from Net
        .DATA[0].7   // Input Letoff A VFD At Reference
        .DATA[1]   // Input Letoff A VFD Speed
        .DATA[2]   // Input Letoff A VFD Amps
        .DATA[3]   // Input Letoff A VFD Max Hertz
        .DATA[4]   // Input Letoff A VFD Motor Nameplate Hertz
        .DATA[5]   // Input Letoff A VFD Motor Nameplate RPM
   p29r16_timer_fault : TIMER[10] := ([2].PRE := 2000, [6].PRE := 3000);   // Winder Winder B VFD Fault Dell Timer
   p29r16_timer_warning : TIMER[4] := ([0].PRE := 10000, [0].ACC := 10020, [0].EN := 1, [0].DN := 1, [1].PRE := 10000, [2].PRE := 10000);   // Winder Winder B VFD Warning Dell Timer
   p29r16_torque_acc_rate : REAL := 0.05;
   p29r16_torque_boost_acc_rate : REAL := 5000.0;
   p29r16_torque_boost_dec_rate : REAL := 2.0;
   p29r16_torque_boost_ref : REAL := 90.0;   // Winder Winder A VFD Request Jog REV
   p29r16_torque_boost_timer : TIMER := (PRE := 500);   // Zone 1 Exhaust VFD PB: Auto Stop
   p29r16_torque_dec_rate : REAL := 0.05;
   p29r16_torque_fast_acc_rate : REAL := 0.8;
   p29r16_torque_fast_dec_rate : REAL := 1.6;
   p29r16_torque_high_ref : REAL := 100.0;
   p29r16_torque_low_ref : REAL := 1.0;
   p29r16_torque_mode_acc_rate : REAL := 5000.0;
   p29r16_torque_mode_dec_rate : REAL := 4.0;
   p29r16_torque_ramp : SYS_ACC_DEC_RAMP := (IN_param_master_accel_rate := 0.05, IN_param_master_decel_rate := 0.05, IN_last_scan_s := 0.032584);
   p29r16_torque_soak_acc_rate : REAL := 0.05;
   p29r16_torque_soak_dec_rate : REAL := 0.05;
   p29r16_torque_start_timer : TIMER := (PRE := 200);   // Timer Winder B Torque Start Timer
   p29r16_vfd_start_request : BOOL;
   p29r16_wdrb_accel_decel : SYS_ACC_DEC_RAMP := (IN_param_master_accel_rate := 25.0, IN_param_master_decel_rate := 25.0, IN_last_scan_s := 0.032442);   // Winder Winder B VFD Accel Decel Ramp
   p29r16_wdrb_active : BOOL;   // Winder Winder B VFD Active
   p29r16_wdrb_ramped_speed : REAL;   // Winder Winder B VFD Ramped Speed
   p29r16_zero_speed : BOOL := 1;   // Winder Winder A VFD At Zero BSpeed
   p29r17 : routine := (comment := -1073741777);   // Winder Winder A Diameter
        .FAULT   // Winder Winder Turret VFD
        .UNACK_FAULT   // Winder Winder A Diameter Unacknowleged Faults Exist
        .UNACK_WARNING   // Winder Winder A Diameter Unacknowleged Warnings Exist
   p29r17_ave_control : CONTROL := (LEN := 19);   // Winder Winder A Diameter Calculation AVE Control
   p29r17_diameter_clac_active : BOOL;   // Winder Winder A Diameter Calculation Calc Active
   p29r17_selected_core_diameter : REAL := 3.25;   // Winder Winder A Diameter Calculation Selected Core Diameter
   p29r17_stack_ctrl : CONTROL := (LEN := 20, POS := 19);   // Winder Winder A Diameter Calculation Stack Control
   p29r17_timer : TIMER[5] := ([0].PRE := 20000, [1].PRE := 500);   // Winder Winder A Diameter Calculation Timers
        [1]   // Winder Winder A Diameter Calculation Sample Timer
   p29r17_timer_fault : TIMER[4];   // Winder Winder A Diameter Calculation Fault Dwell Timer
   p29r17_timer_warning : TIMER[4];   // Winder Winder A Diameter Calculation Warning Dwell Timer
   p29r17_web_speed_at_winder : REAL;   // Winder Winder A Diameter True Web Speed at the Winder Line Speed plus Accumulator Payout [fpm]
   p29r17_winder_a_actual_diam_inch : REAL := 3.25;   // Winder Winder A Diameter Calculation Actual Diameter [in]
   p29r17_winder_a_avg_diam_inch : REAL := 3.25;   // Winder Winder A Diameter Calculation Winder A Average Diameter [in]
   p29r17_winder_a_calc_diam_inch : REAL := 3.25;   // Winder Winder A Diameter Calculated Diameter Inch
   p29r17_winder_a_diam_avg_stack : REAL[1000] := ([0] := 3.25, [1] := 3.25, [2] := 3.25, [3] := 3.25, [4] := 3.25, [5] := 3.25, [6] := 3.25, [7] := 3.25, [8] := 3.25, [9] := 3.25, [10] := 3.25, [11] := 3.25, [12] := 3.25, [13] := 3.25, [14] := 3.25, [15] := 3.25, [16] := 3.25, [17] := 3.25, [18] := 3.25, [19] := 3.25, [20] := 3.25, [21] := 3.25, [22] := 3.25, [23] := 3.25, [24] := 3.25, [25] := 3.25, [26] := 3.25, [27] := 3.25, [28] := 3.25, [29] := 3.25, [30] := 3.25, [31] := 3.25, [32] := 3.25, [33] := 3.25, [34] := 3.25, [35] := 3.25, [36] := 3.25, [37] := 3.25, [38] := 3.25, [39] := 3.25, [40] := 3.25, [41] := 3.25, [42] := 3.25, [43] := 3.25, [44] := 3.25, [45] := 3.25, [46] := 3.25, [47] := 3.25, [48] := 3.25, [49] := 3.25, [50] := 3.25, [51] := 3.25, [52] := 3.25, [53] := 3.25, [54] := 3.25, [55] := 3.25, [56] := 3.25, [57] := 3.25, [58] := 3.25, [59] := 3.25,
        [60] := 3.25, [61] := 3.25, [62] := 3.25, [63] := 3.25, [64] := 3.25, [65] := 3.25, [66] := 3.25, [67] := 3.25, [68] := 3.25, [69] := 3.25, [70] := 3.25, [71] := 3.25, [72] := 3.25, [73] := 3.25, [74] := 3.25, [75] := 3.25, [76] := 3.25, [77] := 3.25, [78] := 3.25, [79] := 3.25, [80] := 3.25, [81] := 3.25, [82] := 3.25, [83] := 3.25, [84] := 3.25, [85] := 3.25, [86] := 3.25, [87] := 3.25, [88] := 3.25, [89] := 3.25, [90] := 3.25, [91] := 3.25, [92] := 3.25, [93] := 3.25, [94] := 3.25, [95] := 3.25, [96] := 3.25, [97] := 3.25, [98] := 3.25, [99] := 3.25, [100] := 3.25, [101] := 3.25, [102] := 3.25, [103] := 3.25, [104] := 3.25, [105] := 3.25, [106] := 3.25, [107] := 3.25, [108] := 3.25, [109] := 3.25, [110] := 3.25, [111] := 3.25, [112] := 3.25, [113] := 3.25, [114] := 3.25, [115] := 3.25, [116] := 3.25, [117] := 3.25, [118] := 3.25, [119] := 3.25,
        [120] := 3.25, [121] := 3.25, [122] := 3.25, [123] := 3.25, [124] := 3.25, [125] := 3.25, [126] := 3.25, [127] := 3.25, [128] := 3.25, [129] := 3.25, [130] := 3.25, [131] := 3.25, [132] := 3.25, [133] := 3.25, [134] := 3.25, [135] := 3.25, [136] := 3.25, [137] := 3.25, [138] := 3.25, [139] := 3.25, [140] := 3.25, [141] := 3.25, [142] := 3.25, [143] := 3.25, [144] := 3.25, [145] := 3.25, [146] := 3.25, [147] := 3.25, [148] := 3.25, [149] := 3.25, [150] := 3.25, [151] := 3.25, [152] := 3.25, [153] := 3.25, [154] := 3.25, [155] := 3.25, [156] := 3.25, [157] := 3.25, [158] := 3.25, [159] := 3.25, [160] := 3.25, [161] := 3.25, [162] := 3.25, [163] := 3.25, [164] := 3.25, [165] := 3.25, [166] := 3.25, [167] := 3.25, [168] := 3.25, [169] := 3.25, [170] := 3.25, [171] := 3.25, [172] := 3.25, [173] := 3.25, [174] := 3.25, [175] := 3.25, [176] := 3.25, [177] := 3.25, [178] := 3.25, [179] := 3.25,
        [180] := 3.25, [181] := 3.25, [182] := 3.25, [183] := 3.25, [184] := 3.25, [185] := 3.25, [186] := 3.25, [187] := 3.25, [188] := 3.25, [189] := 3.25, [190] := 3.25, [191] := 3.25, [192] := 3.25, [193] := 3.25, [194] := 3.25, [195] := 3.25, [196] := 3.25, [197] := 3.25, [198] := 3.25, [199] := 3.25, [200] := 3.25, [201] := 3.25, [202] := 3.25, [203] := 3.25, [204] := 3.25, [205] := 3.25, [206] := 3.25, [207] := 3.25, [208] := 3.25, [209] := 3.25, [210] := 3.25, [211] := 3.25, [212] := 3.25, [213] := 3.25, [214] := 3.25, [215] := 3.25, [216] := 3.25, [217] := 3.25, [218] := 3.25, [219] := 3.25, [220] := 3.25, [221] := 3.25, [222] := 3.25, [223] := 3.25, [224] := 3.25, [225] := 3.25, [226] := 3.25, [227] := 3.25, [228] := 3.25, [229] := 3.25, [230] := 3.25, [231] := 3.25, [232] := 3.25, [233] := 3.25, [234] := 3.25, [235] := 3.25, [236] := 3.25, [237] := 3.25, [238] := 3.25, [239] := 3.25,
